// TIA Portal project "#13-J1200T(夹紧阀断电延时）" (V17)

(* hardware
DEVICE "S7-1200 station_1"  S7-1200 Station
   slot 0: "Rack_0"  S7-1200 Rack  Rack  V1.0
   slot 1: "PLC_1"  CPU 1215C DC/DC/DC  6ES7 215-1AG40-0XB0  V4.5
   slot 2: "DI 16x24VDC_1"  6ES7 221-1BH32-0XB0  V2.0
   slot 3: "DI 16x24VDC_2"  6ES7 221-1BH32-0XB0  V2.0
   slot 4: "DI 16x24VDC_3"  6ES7 221-1BH32-0XB0  V2.0
   slot 5: "DQ 16x24VDC_1"  SM 1222 DQ16 x 24VDC  6ES7 222-1BH32-0XB0  V2.0
   slot 101: "CM 1243-5"  CM 1243-5  6GK7 243-5DX30-0XE0  V1.3
DEVICE "ET 200SP station_1"  ET 200SP-Station
   slot 0: "机架_0"  Rack  6ES5 710-8MAx1
   slot 0: "IO device_1"  IM 155-6 PN ST  6ES7 155-6AU01-0BN0  V4.2
   slot 1: "DI 16x24VDC ST_1"  DI 16x24VDC ST  6ES7 131-6BH01-0BA0  V0.0
      slot 1: "DI 16x24VDC ST_1"  DI 16x24VDC ST
   slot 2: "DI 16x24VDC ST_6"  DI 16x24VDC ST  6ES7 131-6BH01-0BA0  V0.0
      slot 1: "DI 16x24VDC ST_6"  DI 16x24VDC ST
   slot 3: "DI 16x24VDC ST_5"  DI 16x24VDC ST  6ES7 131-6BH01-0BA0  V0.0
      slot 1: "DI 16x24VDC ST_5"  DI 16x24VDC ST
   slot 4: "DI 16x24VDC ST_4"  DI 16x24VDC ST  6ES7 131-6BH01-0BA0  V0.0
      slot 1: "DI 16x24VDC ST_4"  DI 16x24VDC ST
   slot 5: "DI 16x24VDC ST_3"  DI 16x24VDC ST  6ES7 131-6BH01-0BA0  V0.0
      slot 1: "DI 16x24VDC ST_3"  DI 16x24VDC ST
   slot 6: "DI 16x24VDC ST_2"  DI 16x24VDC ST  6ES7 131-6BH01-0BA0  V0.0
      slot 1: "DI 16x24VDC ST_2"  DI 16x24VDC ST
   slot 7: "DI 16x24VDC ST_7"  DI 16x24VDC ST  6ES7 131-6BH01-0BA0  V0.0
      slot 1: "DI 16x24VDC ST_7"  DI 16x24VDC ST
   slot 8: "DI 16x24VDC ST_8"  DI 16x24VDC ST  6ES7 131-6BH01-0BA0  V0.0
      slot 1: "DI 16x24VDC ST_8"  DI 16x24VDC ST
   slot 9: "DI 16x24VDC ST_9"  DI 16x24VDC ST  6ES7 131-6BH01-0BA0  V0.0
      slot 1: "DI 16x24VDC ST_9"  DI 16x24VDC ST
   slot 10: "DI 16x24VDC ST_10"  DI 16x24VDC ST  6ES7 131-6BH01-0BA0  V0.0
      slot 1: "DI 16x24VDC ST_10"  DI 16x24VDC ST
   slot 11: "DI 16x24VDC ST_11"  DI 16x24VDC ST  6ES7 131-6BH01-0BA0  V0.0
      slot 1: "DI 16x24VDC ST_11"  DI 16x24VDC ST
   slot 12: "DI 16x24VDC ST_12"  DI 16x24VDC ST  6ES7 131-6BH01-0BA0  V0.0
      slot 1: "DI 16x24VDC ST_12"  DI 16x24VDC ST
   slot 13: "DQ 16x24VDC/0.5A ST_2"  DQ 16x24VDC/0.5A ST  6ES7 132-6BH01-0BA0  V0.0
      slot 1: "DQ 16x24VDC/0.5A ST_2"  DQ 16x24VDC/0.5A ST
   slot 14: "DQ 16x24VDC/0.5A ST_1"  DQ 16x24VDC/0.5A ST  6ES7 132-6BH01-0BA0  V0.0
      slot 1: "DQ 16x24VDC/0.5A ST_1"  DQ 16x24VDC/0.5A ST
   slot 15: "服务器模块_1"  Server module  6ES7 193-6PA00-0AA0  V1.1
      slot 1: "服务器模块_1"  Server module
   slot 127: "BA 2xRJ45"  BA 2xRJ45  6ES7 193-6AR00-0AA0  V0.0
      slot 1: "Port_1"  X1 P1 R  6ES7 193-6AR00-0AA0  V0.0
      slot 2: "Port_2"  X1 P2 R  6ES7 193-6AR00-0AA0  V0.0
DEVICE "HMI_1"  TP900 Comfort
   slot 0: "HMI_1"  TP900 Comfort  6AV2 124-0JC01-0AX0  15.1.0.0
   slot 1: "HMI_RT_1"  TP900 Comfort  6AV2 124-0JC01-0AX0  15.1.0.0
   slot 5: "HMI_1.IE_CP_1"  PROFINET Interface  15.0.1.0
      slot 1: "PROFINET Interface_1"  PROFINET Interface
         slot 1: "Port_1"  Port
         slot 2: "Port_2"  Port
   slot 7: "HMI_1.MPI/DP_CP_1"  MPI/DP Interface  15.0.1.0
DEVICE "GSD device_2"  GSD.Device
   slot 0: "机架_0"  Rail
   slot 0: "HENGLIANGBIANMAQI"  P+F  Encoder  4.0
DEVICE "GSD device_1"  GSD.Device
   slot 0: "机架_0"  Rail
   slot 0: "滑块站"  P+F  Encoder  4.0
*)

// ===== PLC "PLC_1"  CPU 1215C DC/DC/DC =====

VAR_GLOBAL   // PLC tag table "默认变量表"
   "Tag_1" AT %I0.0 : Bool;
   "Tag_2" AT %I0.1 : Bool;
   "Tag_3" AT %I0.2 : Bool;
   "Tag_4" AT %I0.3 : Bool;
   "Tag_5" AT %I0.4 : Bool;
   "Tag_6" AT %I0.5 : Bool;
   "Tag_7" AT %I0.6 : Bool;
   "Tag_8" AT %I0.7 : Bool;
   "Tag_9" AT %I1.0 : Bool;
   "Tag_10" AT %I1.1 : Bool;
   "Tag_11" AT %I1.2 : Bool;
   "Tag_12" AT %I1.3 : Bool;
   "Tag_13" AT %I1.4 : Bool;
   "Tag_14" AT %I1.5 : Bool;
   "润滑空开" AT %I2.0 : Bool;
   "润滑电机1过载" AT %I2.1 : Bool;
   "Tag_17" AT %I2.4 : Bool;
   "急停KA12" AT %I2.5 : Bool;
   "双阀反馈1" AT %I2.6 : Bool;
   "双阀故障" AT %I3.2 : Bool;
   "滑块空开" AT %I3.3 : Bool;
   "滑块调整防粘连" AT %I3.4 : Bool;
   "Tag_23" AT %I3.5 : Bool;
   "气垫调整空开" AT %I3.6 : Bool;
   "润滑电机2过载_" AT %I2.2 : Bool;
   "润滑电机3过载_" AT %I2.3 : Bool;
   "双阀反馈2" AT %I2.7 : Bool;
   "双阀反馈3" AT %I3.0 : Bool;
   "双阀反馈4" AT %I3.1 : Bool;
   "气垫调整防粘连" AT %I3.7 : Bool;
   "右栅栏空开" AT %I4.0 : Bool;
   "栅栏空开防粘连" AT %I4.1 : Bool;
   "安全栓" AT %I4.2 : Bool;
   "油箱加热触点" AT %I4.3 : Bool;
   "电柜冷却触点" AT %I4.4 : Bool;
   "电机风机启动" AT %I4.5 : Bool;
   "Tag_21" AT %I4.6 : Bool;
   "Tag_22" AT %I4.7 : Bool;
   "Tag_23(1)" AT %I5.0 : Bool;
   "Tag_24" AT %I5.1 : Bool;
   "Tag_25" AT %I5.2 : Bool;
   "Tag_26" AT %I5.3 : Bool;
   "Tag_27" AT %I5.4 : Bool;
   "Tag_28" AT %I5.5 : Bool;
   "Tag_29" AT %I5.6 : Bool;
   "Tag_30" AT %I5.7 : Bool;
   "Tag_31" AT %I6.0 : Bool;
   "Tag_32" AT %I6.1 : Bool;
   "Tag_33" AT %I6.2 : Bool;
   "Tag_34" AT %I6.3 : Bool;
   "Tag_35" AT %I6.4 : Bool;
   "Tag_36" AT %I6.5 : Bool;
   "Tag_37" AT %I6.6 : Bool;
   "Tag_38" AT %I6.7 : Bool;
   "Tag_39" AT %I7.0 : Bool;
   "Tag_40" AT %I7.1 : Bool;
   "Tag_41" AT %I7.2 : Bool;
   "Tag_42" AT %I7.3 : Bool;
   "Tag_43" AT %I7.4 : Bool;
   "Tag_44" AT %I7.5 : Bool;
   "Tag_45" AT %I7.6 : Bool;
   "Tag_46" AT %I7.7 : Bool;
   "气垫手动润滑" AT %I10.0 : Bool;
   "平衡缸手动润滑" AT %I10.1 : Bool;
   "润滑电机启动" AT %I10.2 : Bool;
   "润滑电机停止" AT %I10.3 : Bool;
   "主电机停止" AT %I10.4 : Bool;
   "主电机启动" AT %I10.5 : Bool;
   "微调正反" AT %I10.6 : Bool;
   "微调开动" AT %I10.7 : Bool;
   "气垫调整" AT %I11.0 : Bool;
   "滑块调整" AT %I11.1 : Bool;
   "行程" AT %I11.2 : Bool;
   "模具更换" AT %I11.3 : Bool;
   "微调(1)" AT %I11.4 : Bool;
   "连续" AT %I11.5 : Bool;
   "单次" AT %I11.6 : Bool;
   "寸动" AT %I11.7 : Bool;
   "数据编辑" AT %I12.0 : Bool;
   "寸动1" AT %I12.1 : Bool;
   "寸动2" AT %I12.2 : Bool;
   "连续预置" AT %I12.3 : Bool;
   "停上死点" AT %I12.4 : Bool;
   "故障复位" AT %I12.5 : Bool;
   "液压保护实验" AT %I12.6 : Bool;
   "液压保护重调" AT %I12.7 : Bool;
   "滑块向上" AT %I13.0 : Bool;
   "滑块向下" AT %I13.1 : Bool;
   "滑块调整手动/自动" AT %I13.2 : Bool;
   "模具夹紧/松开" AT %I13.3 : Bool;
   "工作台夹紧/放松" AT %I13.4 : Bool;
   "备用(1)" AT %I13.5 : Bool;
   "油箱加热启动" AT %I13.6 : Bool;
   "油箱加热停止" AT %I13.7 : Bool;
   "平衡缸压力手动/自动" AT %I14.0 : Bool;
   "气垫压力手动/自动" AT %I14.1 : Bool;
   "气垫快排" AT %I14.2 : Bool;
   "气垫调整手动/自动" AT %I14.3 : Bool;
   "气垫向上" AT %I14.4 : Bool;
   "气垫向下" AT %I14.5 : Bool;
   "安全栅栏向上" AT %I14.6 : Bool;
   "安全栅栏向下" AT %I14.7 : Bool;
   "低油位" AT %I15.0 : Bool;
   "高油位" AT %I15.1 : Bool;
   "低油压1" AT %I15.2 : Bool;
   "低油压2" AT %I15.3 : Bool;
   "低油压3" AT %I15.4 : Bool;
   "高油压1" AT %I15.5 : Bool;
   "高油压2" AT %I15.6 : Bool;
   "高油压3" AT %I15.7 : Bool;
   "左前移动闭点1" AT %I16.0 : Bool;
   "左前移动闭点2" AT %I16.1 : Bool;
   "左前移动开点" AT %I16.2 : Bool;
   "左前移动检测" AT %I16.3 : Bool;
   "左后移动闭点1" AT %I16.4 : Bool;
   "左后移动闭点2" AT %I16.5 : Bool;
   "左后移动开点" AT %I16.6 : Bool;
   "左后移动检测" AT %I16.7 : Bool;
   "右前移动短接1" AT %I17.0 : Bool;
   "右前移动短接2" AT %I17.1 : Bool;
   "右前移动短接3" AT %I17.2 : Bool;
   "右前移动短接4" AT %I17.3 : Bool;
   "右后移动短接1" AT %I17.4 : Bool;
   "右后移动短接2" AT %I17.5 : Bool;
   "右后移动短接3" AT %I17.6 : Bool;
   "右后移动短接4" AT %I17.7 : Bool;
   "备用" AT %I18.0 : Bool;
   "梯子开关" AT %I18.1 : Bool;
   "飞轮制动1" AT %I18.2 : Bool;
   "飞轮制动2" AT %I18.3 : Bool;
   "温度保护" AT %I18.4 : Bool;
   "主接触器" AT %I18.5 : Bool;
   "磁场电源" AT %I18.6 : Bool;
   "同步电源" AT %I18.7 : Bool;
   "装置风扇" AT %I19.0 : Bool;
   "风机" AT %I19.1 : Bool;
   "装置正常" AT %I19.2 : Bool;
   "电流保护" AT %I19.3 : Bool;
   "气垫润滑高压" AT %I19.4 : Bool;
   "过滤器堵塞1" AT %I19.5 : Bool;
   "过滤器堵塞2" AT %I19.6 : Bool;
   "过滤器堵塞3" AT %I19.7 : Bool;
   "润滑检测1" AT %I20.0 : Bool;
   "润滑检测2" AT %I20.1 : Bool;
   "润滑检测3" AT %I20.2 : Bool;
   "润滑检测4" AT %I20.3 : Bool;
   "润滑检测5" AT %I20.4 : Bool;
   "润滑检测6" AT %I20.5 : Bool;
   "润滑检测7" AT %I20.6 : Bool;
   "润滑检测8" AT %I20.7 : Bool;
   "润滑检测9" AT %I21.0 : Bool;
   "备用(2)" AT %I21.1 : Bool;
   "离合器压力" AT %I21.2 : Bool;
   "制动器压力" AT %I21.3 : Bool;
   "凸轮1" AT %I21.4 : Bool;
   "凸轮2" AT %I21.5 : Bool;
   "凸轮3" AT %I21.6 : Bool;
   "凸轮4" AT %I21.7 : Bool;
   "灯测试" AT %I22.0 : Bool;
   "蜂鸣器按钮" AT %I22.1 : Bool;
   "自动化气源测试" AT %I22.2 : Bool;
   "Tag_146" AT %I22.3 : Bool;
   "液压保护压力" AT %I22.4 : Bool;
   "卸荷限位" AT %I22.5 : Bool;
   "Tag_149" AT %I22.6 : Bool;
   "滑块上限" AT %I22.7 : Bool;
   "滑块下限" AT %I23.0 : Bool;
   "滑块调整过扭矩" AT %I23.1 : Bool;
   "Tag_153" AT %I23.2 : Bool;
   "Tag_154" AT %I23.3 : Bool;
   "气垫上限" AT %I23.4 : Bool;
   "气垫下限" AT %I23.5 : Bool;
   "Tag_157" AT %I23.6 : Bool;
   "Tag_158" AT %I23.7 : Bool;
   "Tag_159" AT %I24.0 : Bool;
   "Tag_160" AT %I24.1 : Bool;
   "安全栅栏上限位" AT %I24.2 : Bool;
   "安全栅栏下限位" AT %I24.3 : Bool;
   "气垫落到位" AT %I24.4 : Bool;
   "温度开关" AT %I24.5 : Bool;
   "工作台夹紧" AT %I24.6 : Bool;
   "工作台放松" AT %I24.7 : Bool;
   "Tag_167" AT %I25.0 : Bool;
   "平衡缸压力" AT %I25.1 : Bool;
   "工作台夹紧压力" AT %I25.2 : Bool;
   "工作台放松压力" AT %I25.3 : Bool;
   "Tag_171" AT %I25.4 : Bool;
   "Tag_172" AT %I25.5 : Bool;
   "Tag_173" AT %I25.6 : Bool;
   "Tag_174" AT %I25.7 : Bool;
   "Tag_175" AT %I26.0 : Bool;
   "Tag_176" AT %I26.1 : Bool;
   "工作台前落到位" AT %I26.2 : Bool;
   "工作台后落到位" AT %I26.3 : Bool;
   "光电保护开" AT %I26.4 : Bool;
   "光电保护1" AT %I26.5 : Bool;
   "光电保护2" AT %I26.6 : Bool;
   "光电保护3" AT %I26.7 : Bool;
   "光电保护4" AT %I27.0 : Bool;
   "高度保护复位" AT %I27.1 : Bool;
   "防重复3231" AT %I27.2 : Bool;
   "防重复检测3232" AT %I27.3 : Bool;
   "吨位监控" AT %I27.5 : Bool;
   "光电保护角度3235" AT %I27.6 : Bool;
   "Tag_190" AT %I27.7 : Bool;
   "Tag_191" AT %I28.0 : Bool;
   "Tag_192" AT %I28.1 : Bool;
   "Tag_193" AT %I28.2 : Bool;
   "Tag_194" AT %I28.3 : Bool;
   "Tag_195" AT %I28.4 : Bool;
   "Tag_196" AT %I28.5 : Bool;
   "Tag_197" AT %I28.6 : Bool;
   "Tag_198" AT %I28.7 : Bool;
   "Tag_199" AT %I29.0 : Bool;
   "Tag_200" AT %I29.1 : Bool;
   "Tag_201" AT %I29.2 : Bool;
   "Tag_202" AT %I29.3 : Bool;
   "Tag_203" AT %I29.4 : Bool;
   "Tag_204" AT %I29.5 : Bool;
   "Tag_205" AT %I29.6 : Bool;
   "Tag_206" AT %I29.7 : Bool;
   "Tag_207" AT %I30.0 : Bool;
   "Tag_208" AT %I30.1 : Bool;
   "Tag_209" AT %I30.2 : Bool;
   "Tag_210" AT %I30.3 : Bool;
   "Tag_211" AT %I30.4 : Bool;
   "Tag_212" AT %I30.5 : Bool;
   "Tag_213" AT %I30.6 : Bool;
   "Tag_214" AT %I30.7 : Bool;
   "Tag_215" AT %I31.0 : Bool;
   "Tag_216" AT %I31.1 : Bool;
   "Tag_217" AT %I31.2 : Bool;
   "Tag_218" AT %I31.3 : Bool;
   "Tag_219" AT %I31.4 : Bool;
   "Tag_220" AT %I31.5 : Bool;
   "Tag_221" AT %I31.6 : Bool;
   "Tag_222" AT %I31.7 : Bool;
   "Tag_223" AT %I32.0 : Bool;
   "Tag_224" AT %I32.1 : Bool;
   "Tag_225" AT %I32.2 : Bool;
   "Tag_226" AT %I32.3 : Bool;
   "Tag_227" AT %I32.4 : Bool;
   "Tag_228" AT %I32.5 : Bool;
   "Tag_229" AT %I32.6 : Bool;
   "Tag_230" AT %I32.7 : Bool;
   "Tag_231" AT %I33.0 : Bool;
   "Tag_232" AT %I33.1 : Bool;
   "Tag_233" AT %I33.2 : Bool;
   "Tag_234" AT %I33.3 : Bool;
   "Tag_235" AT %I33.4 : Bool;
   "Tag_236" AT %I33.5 : Bool;
   "Tag_237" AT %I33.6 : Bool;
   "Tag_238" AT %I33.7 : Bool;
   "横梁编码器" AT %ID68 : DWord;
   "滑块编码器" AT %ID72 : DInt;
   "Tag_15" AT %Q0.0 : Bool;
   "Tag_16" AT %Q0.1 : Bool;
   "Tag_17(1)" AT %Q0.2 : Bool;
   "Tag_18" AT %Q0.3 : Bool;
   "Tag_19" AT %Q0.4 : Bool;
   "Tag_20" AT %Q0.5 : Bool;
   "Tag_21(1)" AT %Q0.6 : Bool;
   "Tag_22(1)" AT %Q0.7 : Bool;
   "Tag_23(2)" AT %Q1.0 : Bool;
   "Tag_24(1)" AT %Q1.1 : Bool;
   "KA8主电机主接触器" AT %Q2.0 : Bool;
   "KA9主电机正转启动" AT %Q2.1 : Bool;
   "KA10" AT %Q2.2 : Bool;
   "KA11" AT %Q2.3 : Bool;
   "KA12" AT %Q2.4 : Bool;
   "润滑启动(1)" AT %Q2.5 : Bool;
   "气垫调整防粘连(1)" AT %Q2.6 : Bool;
   "气垫向上(2)" AT %Q2.7 : Bool;
   "气垫向下(2)" AT %Q3.0 : Bool;
   "右栅栏防粘连(1)" AT %Q3.1 : Bool;
   "右栅栏向上(1)" AT %Q3.2 : Bool;
   "右栅栏向下(1)" AT %Q3.3 : Bool;
   "润滑油加热(1)" AT %Q3.4 : Bool;
   "滑块调整防粘连(2)" AT %Q3.5 : Bool;
   "滑块向上调整(1)" AT %Q3.6 : Bool;
   "滑块向下调整(1)" AT %Q3.7 : Bool;
   "上死点指示(1)" AT %Q10.0 : Bool;
   "模具放松指示" AT %Q10.1 : Bool;
   "润滑正常指示" AT %Q10.2 : Bool;
   "滤油器堵塞指示" AT %Q10.3 : Bool;
   "油箱油位高指示" AT %Q10.4 : Bool;
   "主电机运行指示" AT %Q10.5 : Bool;
   "液压保护正常指示" AT %Q10.6 : Bool;
   "气垫 落到位指示" AT %Q10.7 : Bool;
   "连续预置指示" AT %Q11.0 : Bool;
   "警铃" AT %Q11.1 : Bool;
   "设备故障指示" AT %Q11.2 : Bool;
   "光电保护指示" AT %Q11.3 : Bool;
   "下死点指示" AT %Q11.4 : Bool;
   "工作台就位夹紧指示" AT %Q11.5 : Bool;
   "工作台放松指示" AT %Q11.6 : Bool;
   "油箱加热指示" AT %Q11.7 : Bool;
   "制动器阀" AT %Q12.0 : Bool;
   "离合器阀1" AT %Q12.1 : Bool;
   "离合器阀2" AT %Q12.2 : Bool;
   "飞轮制动阀" AT %Q12.3 : Bool;
   "平衡缸润滑阀" AT %Q12.4 : Bool;
   "液压保护气源阀" AT %Q12.5 : Bool;
   "液压保护气动泵阀" AT %Q12.6 : Bool;
   "气垫快排阀" AT %Q12.7 : Bool;
   "工作台夹紧阀" AT %Q13.0 : Bool;
   "工作台放松阀" AT %Q13.1 : Bool;
   "气垫润滑阀" AT %Q13.2 : Bool;
   "Tag_95" AT %Q13.3 : Bool;
   "Tag_96" AT %Q13.4 : Bool;
   "Tag_97" AT %Q13.5 : Bool;
   "Tag_98" AT %Q13.6 : Bool;
   "Tag_99" AT %Q13.7 : Bool;
   "Tag_100" AT %Q14.0 : Bool;
   "Tag_101" AT %Q14.1 : Bool;
   "Tag_102" AT %Q14.2 : Bool;
   "Tag_103" AT %Q14.3 : Bool;
   "Tag_104" AT %Q14.4 : Bool;
   "Tag_105" AT %Q14.5 : Bool;
   "Tag_106" AT %Q14.6 : Bool;
   "Tag_107" AT %Q14.7 : Bool;
   "润滑电机过载" AT %M300.0 : Bool;
   "润滑油压低" AT %M300.1 : Bool;
   "润滑高油压" AT %M300.2 : Bool;
   "润滑故障分钟检测" AT %M400.0 : Bool;
   "润滑低油位" AT %M300.3 : Bool;
   "润滑高油位" AT %M300.4 : Bool;
   "润滑故障" AT %M500.0 : Bool;
   "主电机关断延时" AT %M320.1 : Bool;
   "滑块调整条件" AT %M330.0 : Bool;
   "寸动条件1" AT %M7008.0 : Bool;
   "寸动条件2" AT %M7008.1 : Bool;
   "液压保护正常" AT %M7010.0 : Bool;
   "10度" AT %M200.0 : Bool;
   "20度" AT %M200.1 : Bool;
   "30度" AT %M200.2 : Bool;
   "40度" AT %M200.3 : Bool;
   "50" AT %M200.4 : Bool;
   "60" AT %M200.5 : Bool;
   "70" AT %M200.6 : Bool;
   "80" AT %M200.7 : Bool;
   "90" AT %M201.0 : Bool;
   "100" AT %M201.1 : Bool;
   "110" AT %M201.2 : Bool;
   "120" AT %M201.3 : Bool;
   "130" AT %M201.4 : Bool;
   "140" AT %M201.5 : Bool;
   "150" AT %M201.6 : Bool;
   "160" AT %M201.7 : Bool;
   "170" AT %M202.0 : Bool;
   "180" AT %M202.1 : Bool;
   "190" AT %M202.2 : Bool;
   "200" AT %M202.3 : Bool;
   "210" AT %M202.4 : Bool;
   "220" AT %M202.5 : Bool;
   "230" AT %M202.6 : Bool;
   "240" AT %M202.7 : Bool;
   "250" AT %M203.0 : Bool;
   "260" AT %M203.1 : Bool;
   "270" AT %M203.2 : Bool;
   "280" AT %M203.3 : Bool;
   "290" AT %M203.4 : Bool;
   "300" AT %M203.5 : Bool;
   "310" AT %M203.6 : Bool;
   "320" AT %M203.7 : Bool;
   "330" AT %M204.0 : Bool;
   "340" AT %M204.1 : Bool;
   "350" AT %M204.2 : Bool;
   "360" AT %M204.3 : Bool;
   "上死点" AT %M204.4 : Bool;
   "制动监控" AT %M204.5 : Bool;
   "下死点" AT %M204.6 : Bool;
   "单次返回" AT %M204.7 : Bool;
   "光电保护位置" AT %M205.0 : Bool;
   "编码器闭点监控" AT %M14.7 : Bool;
   "单次开始" AT %M14.4 : Bool;
   "编码器开点监控" AT %M15.0 : Bool;
   "编码器故障" AT %M15.1 : Bool;
   "上死点指示" AT %M0.0 : Bool;
   "下死点指示(1)" AT %M0.1 : Bool;
   "滑块软限位上" AT %M15.5 : Bool;
   "上调整设定值" AT %M15.7 : Bool;
   "滑块软限位下" AT %M15.6 : Bool;
   "滑块调整自动向下" AT %M16.1 : Bool;
   "微调反转" AT %M0.2 : Bool;
   "滑块调整自动向上" AT %M16.0 : Bool;
   "滑块调整自动选择" AT %M16.2 : Bool;
   "微调正转" AT %M0.3 : Bool;
   "行程允许" AT %M14.0 : Bool;
   "寸动允许" AT %M14.1 : Bool;
   "寸动开始" AT %M14.2 : Bool;
   "单次允许" AT %M14.3 : Bool;
   "双手开点监测" AT %M11.0 : Bool;
   "双手闭点监测" AT %M11.1 : Bool;
   "急停故障" AT %M6.0 : Bool;
   "润滑次数检测" AT %M11.2 : Bool;
   "润滑频次故障" AT %M11.3 : Bool;
   "单次返回3233" AT %I27.4 : Bool;
   "重复故障" AT %M19.1 : Bool;
   "计数开始" AT %M20.0 : Bool;
   "计数清零" AT %M20.1 : Bool;
   "间歇润滑时间" AT %M19.3 : Bool;
   "Tag_47" AT %MB10 : Byte;
   "Tag_48" AT %MD10 : DWord;
END_VAR

VAR_GLOBAL CONSTANT   // PLC tag table "默认变量表"
   "无(1)" : Pip := 65535;
   "自动更新(1)" : Pip := 0;
   "PIP 1(1)" : Pip := 1;
   "PIP 2(1)" : Pip := 2;
   "PIP 3(1)" : Pip := 3;
   "PIP 4(1)" : Pip := 4;
   "PIP OB 伺服(1)" : Pip := 32768;
   "Local~MC(1)" : Hw_SubModule := 51;
   "Local~Common(1)" : Hw_SubModule := 50;
   "Local~Device(1)" : Hw_Device := 32;
   "Local~Configuration(1)" : Hw_SubModule := 33;
   "Local~Exec(1)" : Hw_SubModule := 52;
   "Local(1)" : Hw_SubModule := 49;
   "Local~PROFINET_接口_1(1)" : Hw_Interface := 64;
   "Local~PROFINET_接口_1~端口_1(1)" : Hw_Interface := 65;
   "Local~HSC_1(1)" : Hw_Hsc := 257;
   "Local~HSC_2(1)" : Hw_Hsc := 258;
   "Local~HSC_3(1)" : Hw_Hsc := 259;
   "Local~HSC_4(1)" : Hw_Hsc := 260;
   "Local~HSC_5(1)" : Hw_Hsc := 261;
   "Local~HSC_6(1)" : Hw_Hsc := 262;
   "Local~AI_2_1" : Hw_SubModule := 263;
   "Local~DI_14_DQ_10_1(1)" : Hw_SubModule := 264;
   "Local~Pulse_1(1)" : Hw_Pwm := 265;
   "Local~Pulse_2(1)" : Hw_Pwm := 266;
   "Local~Pulse_3(1)" : Hw_Pwm := 267;
   "Local~Pulse_4(1)" : Hw_Pwm := 268;
   "Local~CM_1243-5~DP_接口(1)" : Hw_Interface := 269;
   "Local~CM_1243-5(1)" : Hw_SubModule := 271;
   "Local~PROFINET_IO-System(1)" : Hw_IoSystem := 272;
   "Local~DP-Mastersystem(1)" : Hw_IoSystem := 273;
   "Local~DI_16x24VDC_1(1)" : Hw_SubModule := 291;
   "Local~DI_16x24VDC_2(1)" : Hw_SubModule := 292;
   "Local~DQ_16x24VDC_1(1)" : Hw_SubModule := 293;
   "立柱右前操作站~Head" : Hw_Interface := 288;
   "立柱右前操作站~DPSlave" : Hw_DpSlave := 286;
   "立柱右前操作站~DI_32x24VDC_1" : Hw_SubModule := 289;
   "立柱右前操作站~AI_8x12BIT_1" : Hw_SubModule := 294;
   "立柱右前操作站~DI_32x24VDC_2" : Hw_SubModule := 295;
   "立柱右前操作站~DI_32x24VDC_3" : Hw_SubModule := 296;
   "立柱右前操作站~DI_32x24VDC_4" : Hw_SubModule := 297;
   "立柱右前操作站~DO_32x24VDC_0_5A_2" : Hw_SubModule := 299;
   "立柱右前操作站~DO_16x24VDC_0_5A_1" : Hw_SubModule := 290;
   "立柱右前操作站~DI_16x24VDC_1" : Hw_SubModule := 274;
   "横梁站~Head(1)" : Hw_Interface := 280;
   "横梁站~DPSlave(1)" : Hw_DpSlave := 278;
   "横梁站~P+F_Version_2_1_Singleturn_1(1)" : Hw_SubModule := 281;
   "OB_Main(1)" : OB_PCYCLE := 1;
   "OB_Cyclic interrupt" : OB_Cyclic := 30;
   "OB_RackStationFailure" : OB_Any := 86;
   "OB_Startup" : OB_STARTUP := 100;
   "滑块站~Head(1)" : Hw_Interface := 277;
   "滑块站~DPSlave(1)" : Hw_DpSlave := 275;
   "滑块站~32_Bit_Class_2_+_Speed_2_1" : Hw_SubModule := 282;
   "滑块站~32_Bit_Class_2_+_Speed_2_2" : Hw_SubModule := 283;
END_VAR

VAR_GLOBAL   // PLC tag table "变量表_1"
   "主电机启动条件" AT %M800.1 : Bool;
   "产量完成" AT %M800.0 : Bool;
END_VAR

TYPE "用户数据类型_1"
VERSION : 0.1
   STRUCT
      Element_1 : Bool;
   END_STRUCT;
END_TYPE

// folder: 4.1_Line_Operation

TYPE "Operation_Mode"
VERSION : 0.1
   STRUCT
      Auto : Bool;
      Auto_Sim : Bool;
      APC : Bool;
      ATC : Bool;
      Man : Bool;
      Setup : Bool;
      工作模式 : UInt;
      零件表 : UInt;
   END_STRUCT;
END_TYPE

TYPE "4.1_Line_Operation"
VERSION : 0.1
   STRUCT
      Mode_Act : "Operation_Mode";
      Mode_Seting : "Operation_Mode";
      Recipes_Operation : "HMI_Recipe";
      HMI : Array[1..10] of "HMI_State";
   END_STRUCT;
END_TYPE

TYPE "HMI_Recipe"
VERSION : 0.1
   STRUCT
      Recipe : Struct
         Clear : Bool;
         Load : Bool;
         Save : Bool;
         Edit_No : Int;
         Recipe_Edit_Auth : Bool;
         Recipe_Edit_Wizard : Int;
         Load_Active : Bool;
         Save_Active : Bool;
         ii : Int;
         Load_Timer : IEC_TIMER;
         Save_Timer : IEC_TIMER;
      END_STRUCT;
      RecipeExport : Struct
         Done : Bool;
         Busy : Bool;
         Error : Bool;
         Status : Word;
      END_STRUCT;
      RecipeImport : Struct
         Done : Bool;
         Busy : Bool;
         Error : Bool;
         Status : Word;
      END_STRUCT;
   END_STRUCT;
END_TYPE

TYPE "HMI_State"
VERSION : 0.1
   STRUCT
      Command : Struct
         Doub_Part_Dropped_Mem : Bool;
         Part_Dropped_Mem : Bool;
         Part_Picker_Mem : Bool;
         Part_Done_Mem : Bool;
         Optim_Auth : Bool;
         Part_No_Chg_Auth : Bool;
      END_STRUCT;
      State : Struct
         Doub_Part_Dropped_Mem_1 : Bool;
         Part_Dropped_Mem_1 : Bool;
         Part_Picker_Mem_1 : Bool;
         Part_Done_Mem_1 : Bool;
      END_STRUCT;
   END_STRUCT;
END_TYPE

// folder: (top level)

DATA_BLOCK "横梁编码器 _DB"   // DB15
{ S7_Optimized_Access := 'TRUE' }
VERSION : 0.1
   VAR
      "0.0" : Struct
         "+0.0" : DWord;
         "+4.0" : DWord;
         "+8.0" : DWord;
         "+12.0" : DWord;
      END_STRUCT;
      横梁 : Int;
      滑块 : Int;
      滑块_1 : DWord;
      "+0.3" : Int;
      "+0.4" : Int;
      "+0.5" : Int;
      "+0.6" : Int;
      "+0.7" : Int;
   END_VAR
   VAR RETAIN
      "+0.8" : Int;
   END_VAR
   VAR
      "+0.9" : Int;
      "+0.10" : Int;
      "0.11" : Real;
      平衡器分油器检测 : Int;
      横梁分油器检测 : Int;
      滑块分油器检测 : Int;
      气垫分油器检测 : Int;
      "+0.15" : Int;
      "+0.16" : Int;
      "+0.17" : Int;
      "+0.18" : Int;
      "+0.19" : Int;
      "+0.20" : Int;
      "+0.21" : Int;
      "+0.22" : Int;
      "+0.23" : Int;
      "+0.24" : Int;
      "+0.25" : Int;
      "+0.26" : Int;
      "+0.27" : Int;
      "+0.28" : Int;
      "+0.29" : Int;
      "+0.30" : Int;
      平衡器打油次数 : Int;
      主分油器打油次数 : Int;
      滑块打油次数 : Int;
      气点垫打油次数 : Int;
      "+0.35" : Int;
      "+0.36" : Int;
      "+0.37" : Int;
      "+0.38" : Int;
      "+0.39" : Int;
      "+0.40" : Int;
      "+0.41" : Int;
      "+0.42" : Int;
      "+0.43" : Int;
      "+0.44" : Int;
      "+0.45" : Int;
      "+0.46" : Int;
      "+0.47" : Int;
      "+0.48" : Int;
   END_VAR
   VAR RETAIN
      AI : Array[0..10] of DInt;
      D : Array[0..10] of Real;
   END_VAR
   VAR
      AQD : Real;
      产量设定 : Int;
      D107 : Real;
   END_VAR
BEGIN
END_DATA_BLOCK

DATA_BLOCK "滑块编码器_DB"   // DB16
{ S7_Optimized_Access := 'TRUE' }
VERSION : 0.1
   VAR
      "0.0" : Struct
         "+0.0" : DWord;
         "+4.0" : DWord;
         "+8.0" : DWord;
         "+12.0" : DWord;
      END_STRUCT;
      横梁编码器 : Int;
      滑块编码器 : DInt;
      气垫编码器1 : DWord;
      气垫编码器2 : DWord;
      平衡器压力显示_3 : Int;
      电子凸轮编码器 : Int;
      "+0.5" : Real;
      电子凸轮编码器显示 : Int;
      "+0.7" : DInt;
      "+0.8" : Int;
      "+0.9" : Real;
      "+0.10_1" : Int;
      "+0.11" : Int;
      "+0.12" : Int;
      "+0.13" : Int;
      "+0.10" : Int;
      平衡器分油器检测 : Int;
      横梁分油器检测 : Int;
      滑块分油器检测 : Int;
      气垫分油器检测 : Int;
      "+0.15" : Int;
      "+0.16" : Int;
      "+0.17" : Int;
      "+0.18" : Int;
      "+0.19" : Int;
      "+0.20" : Int;
      "+0.21" : Int;
      "+0.22" : Int;
      "+0.23" : Int;
      "+0.24" : Int;
      "+0.25" : Int;
      "+0.26" : Int;
      "+0.27" : Int;
      "+0.28" : Int;
      "+0.29" : Int;
      "+0.30" : Int;
      平衡器打油次数 : Int;
      主分油器打油次数 : Int;
      滑块打油次数 : Int;
      气点垫打油次数 : Int;
      "+0.35" : Int;
      "+0.36" : Int;
      平衡器压力显示_2 : Real;
      平衡器压力显示_1 : Real;
      "+0.39" : Int;
      "+0.40" : Real;
      "+0.41" : Real;
      气垫模拟量 : Int;
      气垫模拟量_1 : Real;
      气垫模拟量_2 : Real;
      "+0.45" : DInt;
      "+0.46" : Int;
      "+0.47" : Real;
      "+0.48" : Int;
   END_VAR
   VAR RETAIN
      AI : Array[0..10] of DInt;
      D : Array[0..20] of Real;
   END_VAR
   VAR
      平衡器压力显示 : Real;
      AQD2 : Real;
      气垫模拟量显示1 : Real;
      气垫模拟量显示2 : Real;
      平衡器设置压力 : Real;
      气垫1压力设置 : Real;
      气垫2压力设置 : Real;
      D100 : Real;
      D101 : Int;
      D102 : Int;
      D103 : Real;
      D104 : Real;
      D105 : Real;
      D106 : Real;
      D107 : Int;
      D108 : Real;
      D109 : Real;
   END_VAR
   VAR RETAIN
      设置产量 : Int;
      当前产量 : Int;
      滑块位置 : Int;
   END_VAR
   VAR
      气垫位置 : Int;
   END_VAR
   VAR RETAIN
      D200 : DInt;
      D201 : Int;
   END_VAR
BEGIN
END_DATA_BLOCK

DATA_BLOCK "计时器"   // DB20
{ S7_Optimized_Access := 'TRUE' }
VERSION : 0.1
   VAR
      润滑检测延时 : IEC_TIMER;
      编码器闭店监控延时 : IEC_TIMER;
      编码器开点监控延时 : IEC_TIMER;
      主电机指示延时 : IEC_TIMER;
      润滑次数检测延时 : IEC_TIMER;
      平衡缸自动润滑计时 : IEC_TIMER;
      气垫自动润滑计时 : IEC_TIMER;
      平衡缸自动润滑间隔 : IEC_TIMER;
      气垫自动润滑间隔 : IEC_TIMER;
      夹紧阀断电延时 : IEC_TIMER;
   END_VAR
BEGIN
END_DATA_BLOCK

DATA_BLOCK "计数器"   // DB21
{ S7_Optimized_Access := 'TRUE' }
VERSION : 0.1
   VAR
      润滑次数检测 : IEC_COUNTER;
   END_VAR
   VAR RETAIN
      产品计数 : IEC_COUNTER;
   END_VAR
BEGIN
END_DATA_BLOCK

DATA_BLOCK "断电保持数据"   // DB30
{ S7_Optimized_Access := 'TRUE' }
VERSION : 0.1
   VAR RETAIN
      当前产量 : Int := 0;
      目标产量 : Int;
   END_VAR
BEGIN
END_DATA_BLOCK

// folder: 04_HMI_Comand_Config

DATA_BLOCK "Line_OP"   // DB10
{ S7_Optimized_Access := 'TRUE' }
VERSION : 0.1
BEGIN
END_DATA_BLOCK

// folder: (top level)

FUNCTION "10-润滑启动" : Void   // FC10, LAD
{ S7_Optimized_Access := 'TRUE' }
VERSION : 0.1
   VAR_TEMP   // added for the SCL form of the ladder/FBD networks
      _w1 : Bool;
   END_VAR
BEGIN

REGION Network 1
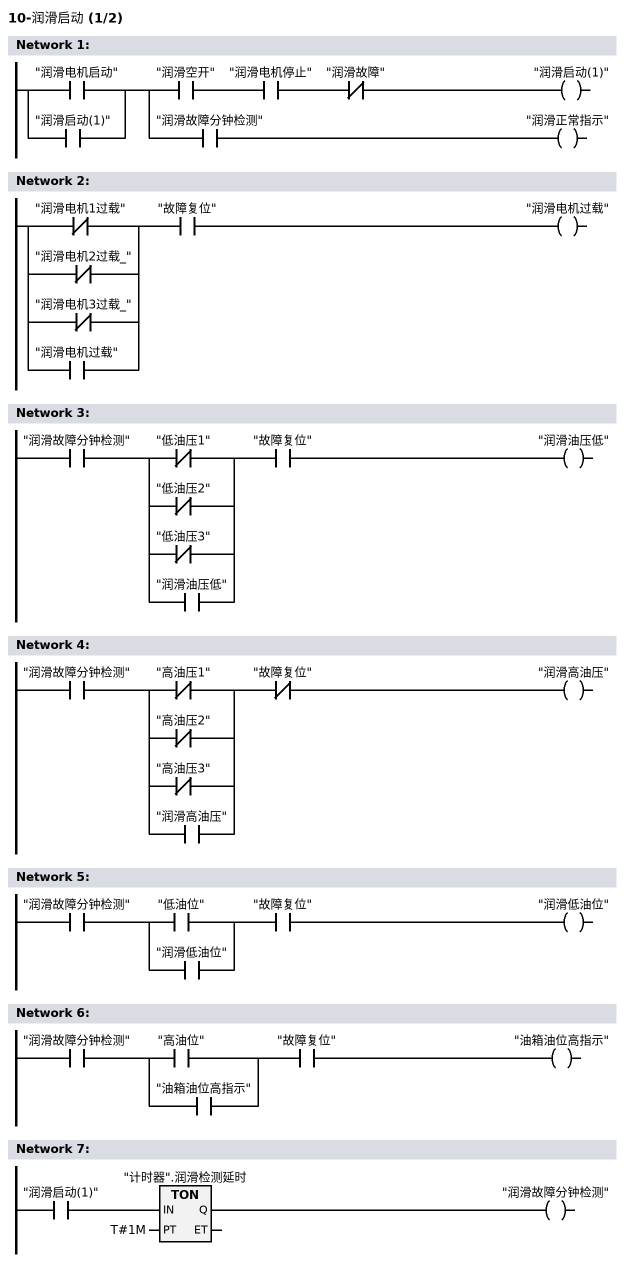
   RUNG wire#powerrail
      Contact( "润滑电机启动" )
      wire#w1
      Contact( "润滑空开" )
      Contact( "润滑电机停止" )
      I_Contact( "润滑故障" )
      Coil( "润滑启动(1)" )
   END_RUNG
   RUNG wire#powerrail
      Contact( "润滑启动(1)" )
   END_RUNG wire#w1
   RUNG wire#w1
      Contact( "润滑故障分钟检测" )
      Coil( "润滑正常指示" )
   END_RUNG
   // the same network as SCL:
   #_w1 := "润滑电机启动" OR "润滑启动(1)";
   "润滑启动(1)" := #_w1 AND "润滑空开" AND "润滑电机停止" AND NOT "润滑故障";
   "润滑正常指示" := #_w1 AND "润滑故障分钟检测";
END_REGION

REGION Network 2
   RUNG wire#powerrail
      I_Contact( "润滑电机1过载" )
      wire#w1
      Contact( "故障复位" )
      Coil( "润滑电机过载" )
   END_RUNG
   RUNG wire#powerrail
      I_Contact( "润滑电机2过载_" )
   END_RUNG wire#w1
   RUNG wire#powerrail
      I_Contact( "润滑电机3过载_" )
   END_RUNG wire#w1
   RUNG wire#powerrail
      Contact( "润滑电机过载" )
   END_RUNG wire#w1
   // the same network as SCL:
   "润滑电机过载" := (NOT "润滑电机1过载" OR NOT "润滑电机2过载_" OR NOT "润滑电机3过载_" OR "润滑电机过载") AND "故障复位";
END_REGION

REGION Network 3
   RUNG wire#powerrail
      Contact( "润滑故障分钟检测" )
      wire#w1
      I_Contact( "低油压1" )
      wire#w2
      Contact( "故障复位" )
      Coil( "润滑油压低" )
   END_RUNG
   RUNG wire#w1
      I_Contact( "低油压2" )
   END_RUNG wire#w2
   RUNG wire#w1
      I_Contact( "低油压3" )
   END_RUNG wire#w2
   RUNG wire#w1
      Contact( "润滑油压低" )
   END_RUNG wire#w2
   // the same network as SCL:
   "润滑油压低" := "润滑故障分钟检测" AND (NOT "低油压1" OR NOT "低油压2" OR NOT "低油压3" OR "润滑油压低") AND "故障复位";
END_REGION

REGION Network 4
   RUNG wire#powerrail
      Contact( "润滑故障分钟检测" )
      wire#w1
      I_Contact( "高油压1" )
      wire#w2
      I_Contact( "故障复位" )
      Coil( "润滑高油压" )
   END_RUNG
   RUNG wire#w1
      I_Contact( "高油压2" )
   END_RUNG wire#w2
   RUNG wire#w1
      I_Contact( "高油压3" )
   END_RUNG wire#w2
   RUNG wire#w1
      Contact( "润滑高油压" )
   END_RUNG wire#w2
   // the same network as SCL:
   "润滑高油压" := "润滑故障分钟检测" AND (NOT "高油压1" OR NOT "高油压2" OR NOT "高油压3" OR "润滑高油压") AND NOT "故障复位";
END_REGION

REGION Network 5
   RUNG wire#powerrail
      Contact( "润滑故障分钟检测" )
      wire#w1
      Contact( "低油位" )
      wire#w2
      Contact( "故障复位" )
      Coil( "润滑低油位" )
   END_RUNG
   RUNG wire#w1
      Contact( "润滑低油位" )
   END_RUNG wire#w2
   // the same network as SCL:
   "润滑低油位" := "润滑故障分钟检测" AND ("低油位" OR "润滑低油位") AND "故障复位";
END_REGION

REGION Network 6
   RUNG wire#powerrail
      Contact( "润滑故障分钟检测" )
      wire#w1
      Contact( "高油位" )
      wire#w2
      Contact( "故障复位" )
      Coil( "油箱油位高指示" )
   END_RUNG
   RUNG wire#w1
      Contact( "油箱油位高指示" )
   END_RUNG wire#w2
   // the same network as SCL:
   "油箱油位高指示" := "润滑故障分钟检测" AND ("高油位" OR "油箱油位高指示") AND "故障复位";
END_REGION

REGION Network 7
   "计时器".润滑检测延时.TON(IN := "润滑启动(1)", PT := T#1M);
   "润滑故障分钟检测" := "计时器".润滑检测延时.Q;
END_REGION

REGION Network 8
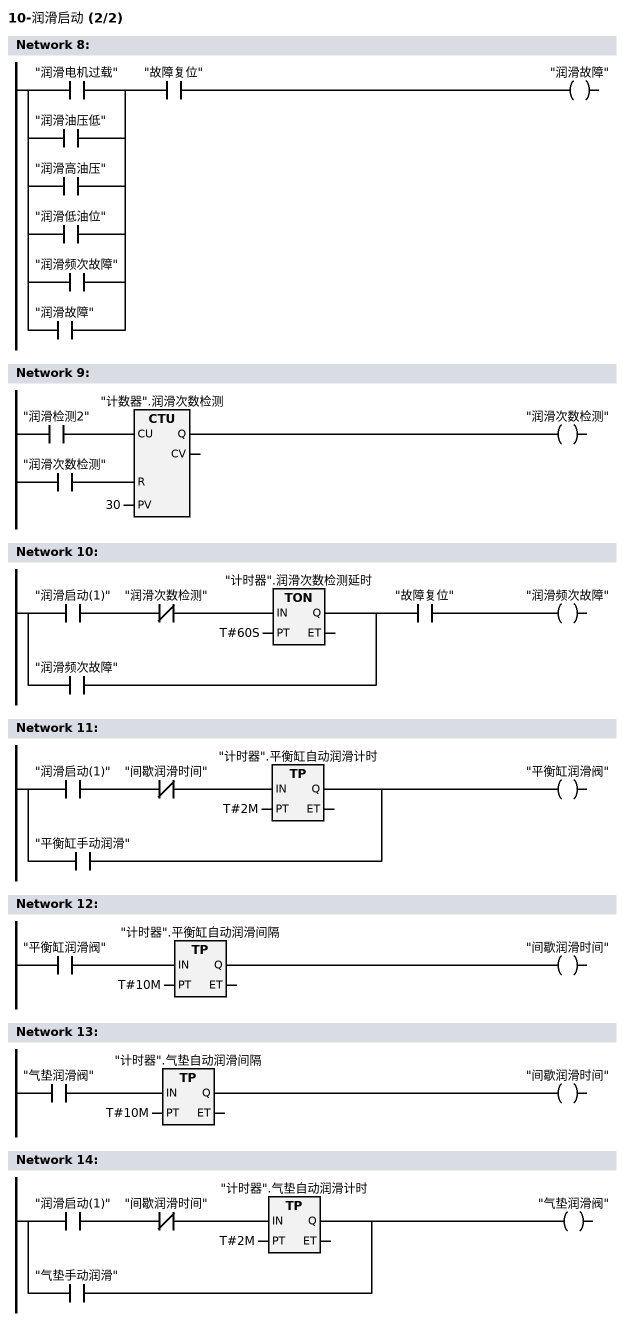
   RUNG wire#powerrail
      Contact( "润滑电机过载" )
      wire#w1
      Contact( "故障复位" )
      Coil( "润滑故障" )
   END_RUNG
   RUNG wire#powerrail
      Contact( "润滑油压低" )
   END_RUNG wire#w1
   RUNG wire#powerrail
      Contact( "润滑高油压" )
   END_RUNG wire#w1
   RUNG wire#powerrail
      Contact( "润滑低油位" )
   END_RUNG wire#w1
   RUNG wire#powerrail
      Contact( "润滑频次故障" )
   END_RUNG wire#w1
   RUNG wire#powerrail
      Contact( "润滑故障" )
   END_RUNG wire#w1
   // the same network as SCL:
   "润滑故障" := ("润滑电机过载" OR "润滑油压低" OR "润滑高油压" OR "润滑低油位" OR "润滑频次故障" OR "润滑故障") AND "故障复位";
END_REGION

REGION Network 9
   "计数器".润滑次数检测.CTU(CU := "润滑检测2", R := "润滑次数检测", PV := 30);
   "润滑次数检测" := "计数器".润滑次数检测.Q;
END_REGION

REGION Network 10
   "计时器".润滑次数检测延时.TON(IN := "润滑启动(1)" AND NOT "润滑次数检测", PT := T#60S);
   "润滑频次故障" := ("计时器".润滑次数检测延时.Q OR "润滑频次故障") AND "故障复位";
END_REGION

REGION Network 11
   "计时器".平衡缸自动润滑计时.TP(IN := "润滑启动(1)" AND NOT "间歇润滑时间", PT := T#2M);
   "平衡缸润滑阀" := "计时器".平衡缸自动润滑计时.Q OR "平衡缸手动润滑";
END_REGION

REGION Network 12
   "计时器".平衡缸自动润滑间隔.TP(IN := "平衡缸润滑阀", PT := T#10M);
   "间歇润滑时间" := "计时器".平衡缸自动润滑间隔.Q;
END_REGION

REGION Network 13
   "计时器".气垫自动润滑间隔.TP(IN := "气垫润滑阀", PT := T#10M);
   "间歇润滑时间" := "计时器".气垫自动润滑间隔.Q;
END_REGION

REGION Network 14
   "计时器".气垫自动润滑计时.TP(IN := "润滑启动(1)" AND NOT "间歇润滑时间", PT := T#2M);
   "气垫润滑阀" := "计时器".气垫自动润滑计时.Q OR "气垫手动润滑";
END_REGION
END_FUNCTION

FUNCTION "20-主电机启动程序" : Void   // FC20, LAD
{ S7_Optimized_Access := 'TRUE' }
VERSION : 0.1
BEGIN

REGION Network 1
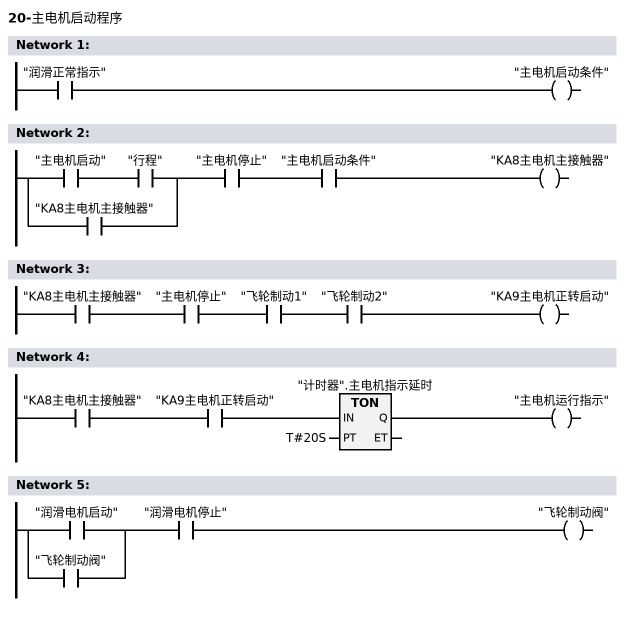
   RUNG wire#powerrail
      Contact( "润滑正常指示" )
      Coil( "主电机启动条件" )
   END_RUNG
   // the same network as SCL:
   "主电机启动条件" := "润滑正常指示";
END_REGION

REGION Network 2
   RUNG wire#powerrail
      Contact( "主电机启动" )
      Contact( "行程" )
      wire#w1
      Contact( "主电机停止" )
      Contact( "主电机启动条件" )
      Coil( "KA8主电机主接触器" )
   END_RUNG
   RUNG wire#powerrail
      Contact( "KA8主电机主接触器" )
   END_RUNG wire#w1
   // the same network as SCL:
   "KA8主电机主接触器" := (("主电机启动" AND "行程") OR "KA8主电机主接触器") AND "主电机停止" AND "主电机启动条件";
END_REGION

REGION Network 3
   RUNG wire#powerrail
      Contact( "KA8主电机主接触器" )
      Contact( "主电机停止" )
      Contact( "飞轮制动1" )
      Contact( "飞轮制动2" )
      Coil( "KA9主电机正转启动" )
   END_RUNG
   // the same network as SCL:
   "KA9主电机正转启动" := "KA8主电机主接触器" AND "主电机停止" AND "飞轮制动1" AND "飞轮制动2";
END_REGION

REGION Network 4
   "计时器".主电机指示延时.TON(IN := "KA8主电机主接触器" AND "KA9主电机正转启动", PT := T#20S);
   "主电机运行指示" := "计时器".主电机指示延时.Q;
END_REGION

REGION Network 5
   RUNG wire#powerrail
      Contact( "润滑电机启动" )
      wire#w1
      Contact( "润滑电机停止" )
      Coil( "飞轮制动阀" )
   END_RUNG
   RUNG wire#powerrail
      Contact( "飞轮制动阀" )
   END_RUNG wire#w1
   // the same network as SCL:
   "飞轮制动阀" := ("润滑电机启动" OR "飞轮制动阀") AND "润滑电机停止";
END_REGION
END_FUNCTION

FUNCTION "30-滑块行程" : Void   // FC30, LAD
{ S7_Optimized_Access := 'TRUE' }
VERSION : 0.1
   VAR_TEMP
      双手闭点检测 : Bool;
   END_VAR
BEGIN

REGION Network 1
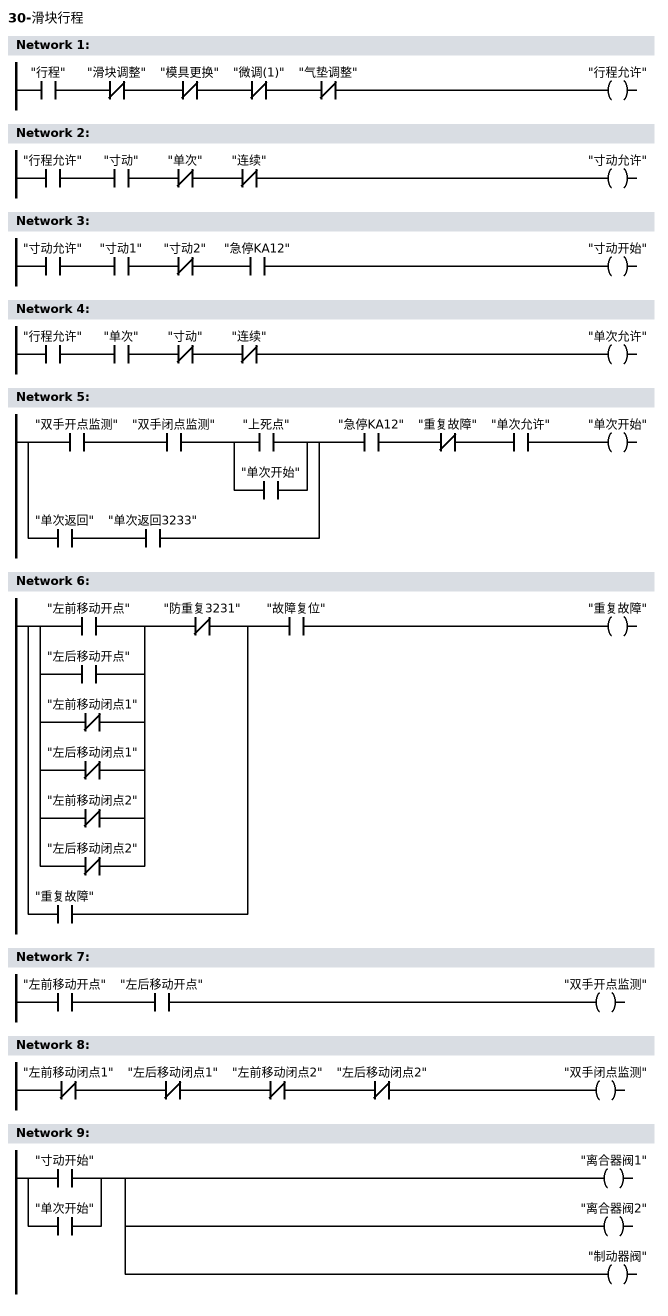
   RUNG wire#powerrail
      Contact( "行程" )
      I_Contact( "滑块调整" )
      I_Contact( "模具更换" )
      I_Contact( "微调(1)" )
      I_Contact( "气垫调整" )
      Coil( "行程允许" )
   END_RUNG
   // the same network as SCL:
   "行程允许" := "行程" AND NOT "滑块调整" AND NOT "模具更换" AND NOT "微调(1)" AND NOT "气垫调整";
END_REGION

REGION Network 2
   RUNG wire#powerrail
      Contact( "行程允许" )
      Contact( "寸动" )
      I_Contact( "单次" )
      I_Contact( "连续" )
      Coil( "寸动允许" )
   END_RUNG
   // the same network as SCL:
   "寸动允许" := "行程允许" AND "寸动" AND NOT "单次" AND NOT "连续";
END_REGION

REGION Network 3
   RUNG wire#powerrail
      Contact( "寸动允许" )
      Contact( "寸动1" )
      I_Contact( "寸动2" )
      Contact( "急停KA12" )
      Coil( "寸动开始" )
   END_RUNG
   // the same network as SCL:
   "寸动开始" := "寸动允许" AND "寸动1" AND NOT "寸动2" AND "急停KA12";
END_REGION

REGION Network 4
   RUNG wire#powerrail
      Contact( "行程允许" )
      Contact( "单次" )
      I_Contact( "寸动" )
      I_Contact( "连续" )
      Coil( "单次允许" )
   END_RUNG
   // the same network as SCL:
   "单次允许" := "行程允许" AND "单次" AND NOT "寸动" AND NOT "连续";
END_REGION

REGION Network 5
   RUNG wire#powerrail
      Contact( "双手开点监测" )
      Contact( "双手闭点监测" )
      wire#w1
      Contact( "上死点" )
      wire#w2
      Contact( "急停KA12" )
      I_Contact( "重复故障" )
      Contact( "单次允许" )
      Coil( "单次开始" )
   END_RUNG
   RUNG wire#w1
      Contact( "单次开始" )
   END_RUNG wire#w2
   RUNG wire#powerrail
      Contact( "单次返回" )
      Contact( "单次返回3233" )
   END_RUNG wire#w2
   // the same network as SCL:
   "单次开始" := (("双手开点监测" AND "双手闭点监测" AND ("上死点" OR "单次开始")) OR ("单次返回" AND "单次返回3233")) AND "急停KA12" AND NOT "重复故障" AND "单次允许";
END_REGION

REGION Network 6
   RUNG wire#powerrail
      Contact( "左前移动开点" )
      wire#w1
      I_Contact( "防重复3231" )
      wire#w2
      Contact( "故障复位" )
      Coil( "重复故障" )
   END_RUNG
   RUNG wire#powerrail
      Contact( "左后移动开点" )
   END_RUNG wire#w1
   RUNG wire#powerrail
      I_Contact( "左前移动闭点1" )
   END_RUNG wire#w1
   RUNG wire#powerrail
      I_Contact( "左后移动闭点1" )
   END_RUNG wire#w1
   RUNG wire#powerrail
      I_Contact( "左前移动闭点2" )
   END_RUNG wire#w1
   RUNG wire#powerrail
      I_Contact( "左后移动闭点2" )
   END_RUNG wire#w1
   RUNG wire#powerrail
      Contact( "重复故障" )
   END_RUNG wire#w2
   // the same network as SCL:
   "重复故障" := ((("左前移动开点" OR "左后移动开点" OR NOT "左前移动闭点1" OR NOT "左后移动闭点1" OR NOT "左前移动闭点2" OR NOT "左后移动闭点2") AND NOT "防重复3231") OR "重复故障") AND "故障复位";
END_REGION

REGION Network 7
   RUNG wire#powerrail
      Contact( "左前移动开点" )
      Contact( "左后移动开点" )
      Coil( "双手开点监测" )
   END_RUNG
   // the same network as SCL:
   "双手开点监测" := "左前移动开点" AND "左后移动开点";
END_REGION

REGION Network 8
   RUNG wire#powerrail
      I_Contact( "左前移动闭点1" )
      I_Contact( "左后移动闭点1" )
      I_Contact( "左前移动闭点2" )
      I_Contact( "左后移动闭点2" )
      Coil( "双手闭点监测" )
   END_RUNG
   // the same network as SCL:
   "双手闭点监测" := NOT "左前移动闭点1" AND NOT "左后移动闭点1" AND NOT "左前移动闭点2" AND NOT "左后移动闭点2";
END_REGION

REGION Network 9
   RUNG wire#powerrail
      Contact( "寸动开始" )
      wire#w1
      Coil( "离合器阀1" )
   END_RUNG
   RUNG wire#powerrail
      Contact( "单次开始" )
   END_RUNG wire#w1
   RUNG wire#w1
      Coil( "离合器阀2" )
   END_RUNG
   RUNG wire#w1
      Coil( "制动器阀" )
   END_RUNG
   // the same network as SCL:
   "离合器阀1" := "寸动开始" OR "单次开始";
   "离合器阀2" := "离合器阀1";
   "制动器阀" := "离合器阀1";
END_REGION
END_FUNCTION

FUNCTION "40-滑块调整程序" : Void   // FC40, LAD
{ S7_Optimized_Access := 'TRUE' }
VERSION : 0.1
BEGIN

REGION Network 1
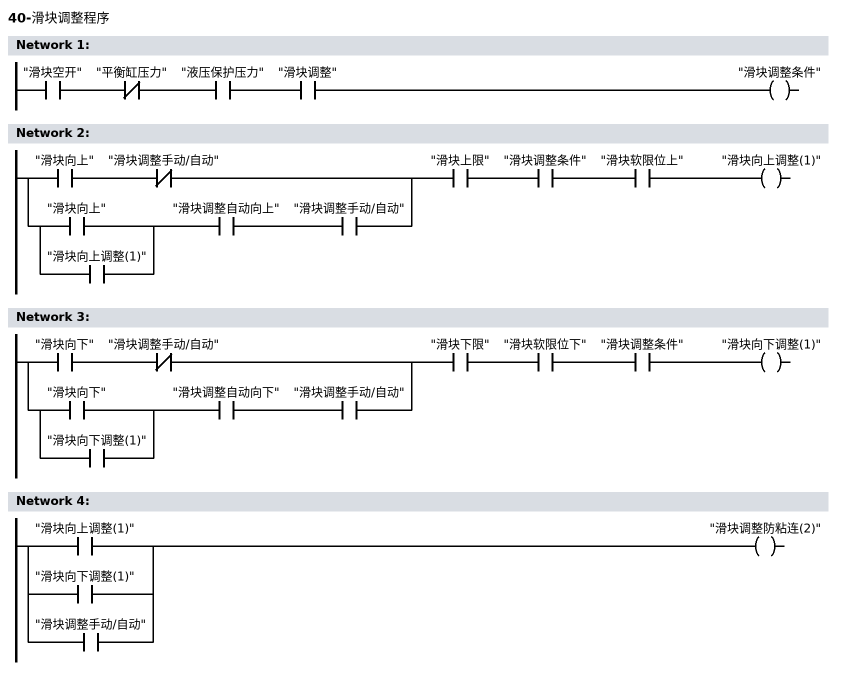
   RUNG wire#powerrail
      Contact( "滑块空开" )
      I_Contact( "平衡缸压力" )
      Contact( "液压保护压力" )
      Contact( "滑块调整" )
      Coil( "滑块调整条件" )
   END_RUNG
   // the same network as SCL:
   "滑块调整条件" := "滑块空开" AND NOT "平衡缸压力" AND "液压保护压力" AND "滑块调整";
END_REGION

REGION Network 2
   RUNG wire#powerrail
      Contact( "滑块向上" )
      I_Contact( "滑块调整手动/自动" )
      wire#w1
      Contact( "滑块上限" )
      Contact( "滑块调整条件" )
      Contact( "滑块软限位上" )
      Coil( "滑块向上调整(1)" )
   END_RUNG
   RUNG wire#powerrail
      Contact( "滑块向上" )
      wire#w2
      Contact( "滑块调整自动向上" )
      Contact( "滑块调整手动/自动" )
   END_RUNG wire#w1
   RUNG wire#powerrail
      Contact( "滑块向上调整(1)" )
   END_RUNG wire#w2
   // the same network as SCL:
   "滑块向上调整(1)" := (("滑块向上" AND NOT "滑块调整手动/自动") OR (("滑块向上" OR "滑块向上调整(1)") AND "滑块调整自动向上" AND "滑块调整手动/自动")) AND "滑块上限" AND "滑块调整条件" AND "滑块软限位上";
END_REGION

REGION Network 3
   RUNG wire#powerrail
      Contact( "滑块向下" )
      I_Contact( "滑块调整手动/自动" )
      wire#w1
      Contact( "滑块下限" )
      Contact( "滑块软限位下" )
      Contact( "滑块调整条件" )
      Coil( "滑块向下调整(1)" )
   END_RUNG
   RUNG wire#powerrail
      Contact( "滑块向下" )
      wire#w2
      Contact( "滑块调整自动向下" )
      Contact( "滑块调整手动/自动" )
   END_RUNG wire#w1
   RUNG wire#powerrail
      Contact( "滑块向下调整(1)" )
   END_RUNG wire#w2
   // the same network as SCL:
   "滑块向下调整(1)" := (("滑块向下" AND NOT "滑块调整手动/自动") OR (("滑块向下" OR "滑块向下调整(1)") AND "滑块调整自动向下" AND "滑块调整手动/自动")) AND "滑块下限" AND "滑块软限位下" AND "滑块调整条件";
END_REGION

REGION Network 4
   RUNG wire#powerrail
      Contact( "滑块向上调整(1)" )
      wire#w1
      Coil( "滑块调整防粘连(2)" )
   END_RUNG
   RUNG wire#powerrail
      Contact( "滑块向下调整(1)" )
   END_RUNG wire#w1
   RUNG wire#powerrail
      Contact( "滑块调整手动/自动" )
   END_RUNG wire#w1
   // the same network as SCL:
   "滑块调整防粘连(2)" := "滑块向上调整(1)" OR "滑块向下调整(1)" OR "滑块调整手动/自动";
END_REGION
END_FUNCTION

FUNCTION "50-移动工作台程序" : Void   // FC50, LAD
{ S7_Optimized_Access := 'TRUE' }
VERSION : 0.1
BEGIN

REGION Network 1
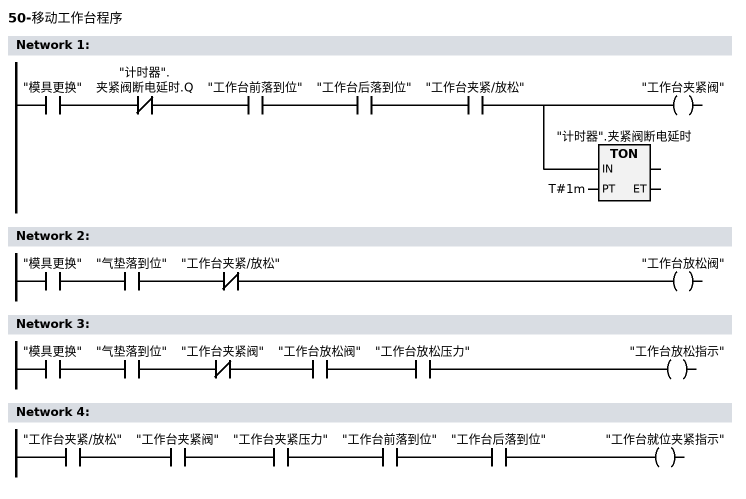
   "工作台夹紧阀" := "模具更换" AND NOT "计时器".夹紧阀断电延时.Q AND "工作台前落到位" AND "工作台后落到位" AND "工作台夹紧/放松";
   "计时器".夹紧阀断电延时.TON(IN := "工作台夹紧阀", PT := T#1m);
END_REGION

REGION Network 2
   RUNG wire#powerrail
      Contact( "模具更换" )
      Contact( "气垫落到位" )
      I_Contact( "工作台夹紧/放松" )
      Coil( "工作台放松阀" )
   END_RUNG
   // the same network as SCL:
   "工作台放松阀" := "模具更换" AND "气垫落到位" AND NOT "工作台夹紧/放松";
END_REGION

REGION Network 3
   RUNG wire#powerrail
      Contact( "模具更换" )
      Contact( "气垫落到位" )
      I_Contact( "工作台夹紧阀" )
      Contact( "工作台放松阀" )
      Contact( "工作台放松压力" )
      Coil( "工作台放松指示" )
   END_RUNG
   // the same network as SCL:
   "工作台放松指示" := "模具更换" AND "气垫落到位" AND NOT "工作台夹紧阀" AND "工作台放松阀" AND "工作台放松压力";
END_REGION

REGION Network 4
   RUNG wire#powerrail
      Contact( "工作台夹紧/放松" )
      Contact( "工作台夹紧阀" )
      Contact( "工作台夹紧压力" )
      Contact( "工作台前落到位" )
      Contact( "工作台后落到位" )
      Coil( "工作台就位夹紧指示" )
   END_RUNG
   // the same network as SCL:
   "工作台就位夹紧指示" := "工作台夹紧/放松" AND "工作台夹紧阀" AND "工作台夹紧压力" AND "工作台前落到位" AND "工作台后落到位";
END_REGION
END_FUNCTION

FUNCTION "60-气垫控制" : Void   // FC60, LAD
{ S7_Optimized_Access := 'TRUE' }
VERSION : 0.1
BEGIN

REGION Network 1
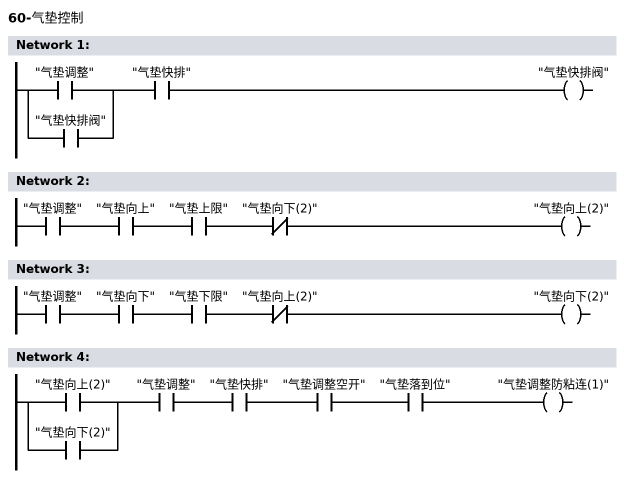
   RUNG wire#powerrail
      Contact( "气垫调整" )
      wire#w1
      Contact( "气垫快排" )
      Coil( "气垫快排阀" )
   END_RUNG
   RUNG wire#powerrail
      Contact( "气垫快排阀" )
   END_RUNG wire#w1
   // the same network as SCL:
   "气垫快排阀" := ("气垫调整" OR "气垫快排阀") AND "气垫快排";
END_REGION

REGION Network 2
   RUNG wire#powerrail
      Contact( "气垫调整" )
      Contact( "气垫向上" )
      Contact( "气垫上限" )
      I_Contact( "气垫向下(2)" )
      Coil( "气垫向上(2)" )
   END_RUNG
   // the same network as SCL:
   "气垫向上(2)" := "气垫调整" AND "气垫向上" AND "气垫上限" AND NOT "气垫向下(2)";
END_REGION

REGION Network 3
   RUNG wire#powerrail
      Contact( "气垫调整" )
      Contact( "气垫向下" )
      Contact( "气垫下限" )
      I_Contact( "气垫向上(2)" )
      Coil( "气垫向下(2)" )
   END_RUNG
   // the same network as SCL:
   "气垫向下(2)" := "气垫调整" AND "气垫向下" AND "气垫下限" AND NOT "气垫向上(2)";
END_REGION

REGION Network 4
   RUNG wire#powerrail
      Contact( "气垫向上(2)" )
      wire#w1
      Contact( "气垫调整" )
      Contact( "气垫快排" )
      Contact( "气垫调整空开" )
      Contact( "气垫落到位" )
      Coil( "气垫调整防粘连(1)" )
   END_RUNG
   RUNG wire#powerrail
      Contact( "气垫向下(2)" )
   END_RUNG wire#w1
   // the same network as SCL:
   "气垫调整防粘连(1)" := ("气垫向上(2)" OR "气垫向下(2)") AND "气垫调整" AND "气垫快排" AND "气垫调整空开" AND "气垫落到位";
END_REGION
END_FUNCTION

FUNCTION "70-液压保护" : Void   // FC70, LAD
{ S7_Optimized_Access := 'TRUE' }
VERSION : 0.1
BEGIN

REGION Network 1
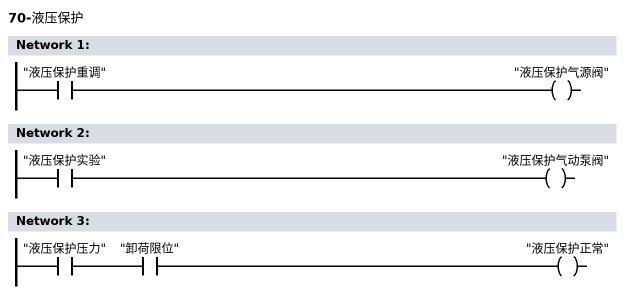
   RUNG wire#powerrail
      Contact( "液压保护重调" )
      Coil( "液压保护气源阀" )
   END_RUNG
   // the same network as SCL:
   "液压保护气源阀" := "液压保护重调";
END_REGION

REGION Network 2
   RUNG wire#powerrail
      Contact( "液压保护实验" )
      Coil( "液压保护气动泵阀" )
   END_RUNG
   // the same network as SCL:
   "液压保护气动泵阀" := "液压保护实验";
END_REGION

REGION Network 3
   RUNG wire#powerrail
      Contact( "液压保护压力" )
      Contact( "卸荷限位" )
      Coil( "液压保护正常" )
   END_RUNG
   // the same network as SCL:
   "液压保护正常" := "液压保护压力" AND "卸荷限位";
END_REGION
END_FUNCTION

FUNCTION "80-产品计数" : Void   // FC80, LAD
{ S7_Optimized_Access := 'TRUE' }
VERSION : 0.1
BEGIN

REGION Network 1
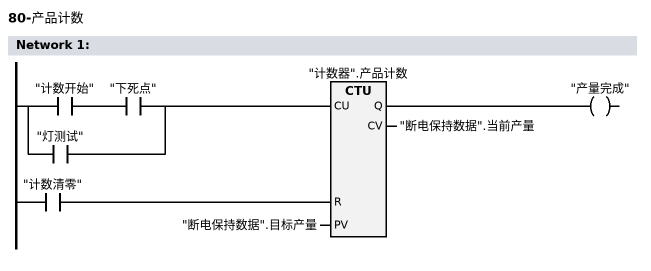
   "计数器".产品计数.CTU(CU := ("计数开始" AND "下死点") OR "灯测试", R := "计数清零", PV := "断电保持数据".目标产量, CV => "断电保持数据".当前产量);
   "产量完成" := "计数器".产品计数.Q;
END_REGION
END_FUNCTION

FUNCTION "横梁编码器调制" : Void   // FC90, LAD
{ S7_Optimized_Access := 'TRUE' }
VERSION : 0.1
BEGIN

REGION Network 1
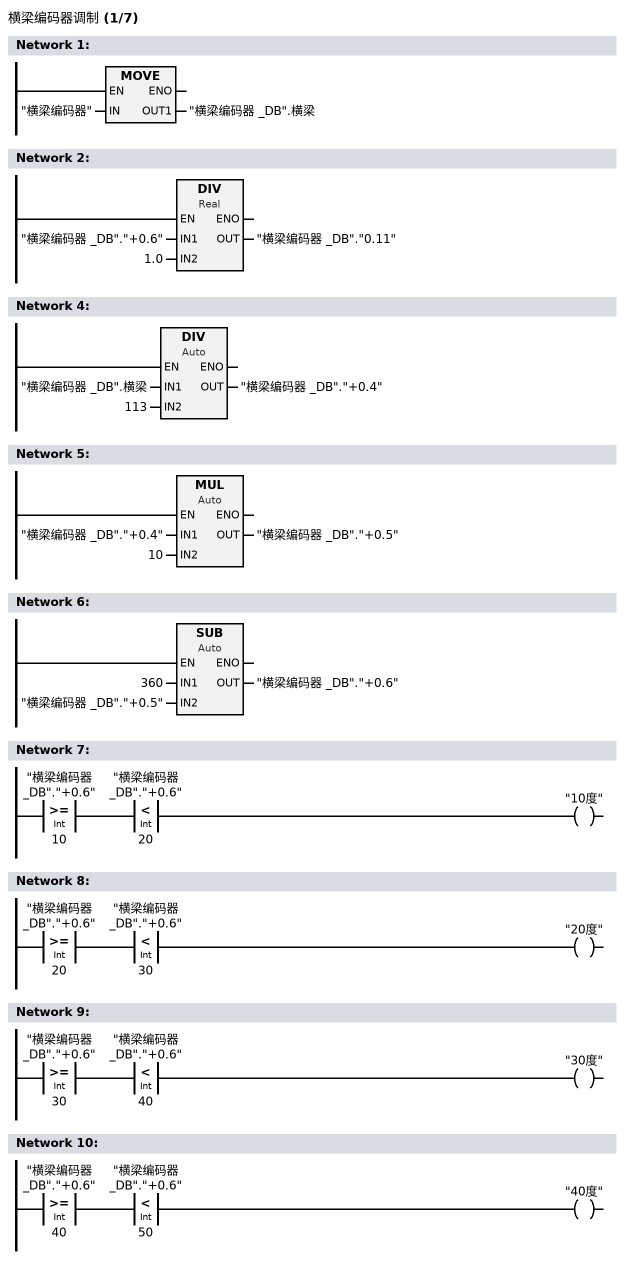
   RUNG wire#powerrail
      Move(in := "横梁编码器", out1 => "横梁编码器 _DB".横梁)
   END_RUNG
   // the same network as SCL:
   "横梁编码器 _DB".横梁 := "横梁编码器";
END_REGION

REGION Network 2
   RUNG wire#powerrail
      { S7_Templates := "SrcType := Real" } Div(in1 := "横梁编码器 _DB"."+0.6", in2 := 1.0, out => "横梁编码器 _DB"."0.11")
   END_RUNG
   // the same network as SCL:
   "横梁编码器 _DB"."0.11" := "横梁编码器 _DB"."+0.6" / 1.0;
END_REGION

REGION Network 4
   RUNG wire#powerrail
      Div(in1 := "横梁编码器 _DB".横梁, in2 := 113, out => "横梁编码器 _DB"."+0.4")
   END_RUNG
   // the same network as SCL:
   "横梁编码器 _DB"."+0.4" := "横梁编码器 _DB".横梁 / 113;
END_REGION

REGION Network 5
   RUNG wire#powerrail
      Mul(in1 := "横梁编码器 _DB"."+0.4", in2 := 10, out => "横梁编码器 _DB"."+0.5")
   END_RUNG
   // the same network as SCL:
   "横梁编码器 _DB"."+0.5" := "横梁编码器 _DB"."+0.4" * 10;
END_REGION

REGION Network 6
   RUNG wire#powerrail
      Sub(in1 := 360, in2 := "横梁编码器 _DB"."+0.5", out => "横梁编码器 _DB"."+0.6")
   END_RUNG
   // the same network as SCL:
   "横梁编码器 _DB"."+0.6" := 360 - "横梁编码器 _DB"."+0.5";
END_REGION

REGION Network 7
   RUNG wire#powerrail
      { S7_Templates := "SrcType := Int" } GE_Contact(in1 := "横梁编码器 _DB"."+0.6", in2 := 10)
      { S7_Templates := "SrcType := Int" } LT_Contact(in1 := "横梁编码器 _DB"."+0.6", in2 := 20)
      Coil( "10度" )
   END_RUNG
   // the same network as SCL:
   "10度" := ("横梁编码器 _DB"."+0.6" >= 10) AND ("横梁编码器 _DB"."+0.6" < 20);
END_REGION

REGION Network 8
   RUNG wire#powerrail
      { S7_Templates := "SrcType := Int" } GE_Contact(in1 := "横梁编码器 _DB"."+0.6", in2 := 20)
      { S7_Templates := "SrcType := Int" } LT_Contact(in1 := "横梁编码器 _DB"."+0.6", in2 := 30)
      Coil( "20度" )
   END_RUNG
   // the same network as SCL:
   "20度" := ("横梁编码器 _DB"."+0.6" >= 20) AND ("横梁编码器 _DB"."+0.6" < 30);
END_REGION

REGION Network 9
   RUNG wire#powerrail
      { S7_Templates := "SrcType := Int" } GE_Contact(in1 := "横梁编码器 _DB"."+0.6", in2 := 30)
      { S7_Templates := "SrcType := Int" } LT_Contact(in1 := "横梁编码器 _DB"."+0.6", in2 := 40)
      Coil( "30度" )
   END_RUNG
   // the same network as SCL:
   "30度" := ("横梁编码器 _DB"."+0.6" >= 30) AND ("横梁编码器 _DB"."+0.6" < 40);
END_REGION

REGION Network 10
   RUNG wire#powerrail
      { S7_Templates := "SrcType := Int" } GE_Contact(in1 := "横梁编码器 _DB"."+0.6", in2 := 40)
      { S7_Templates := "SrcType := Int" } LT_Contact(in1 := "横梁编码器 _DB"."+0.6", in2 := 50)
      Coil( "40度" )
   END_RUNG
   // the same network as SCL:
   "40度" := ("横梁编码器 _DB"."+0.6" >= 40) AND ("横梁编码器 _DB"."+0.6" < 50);
END_REGION

REGION Network 11
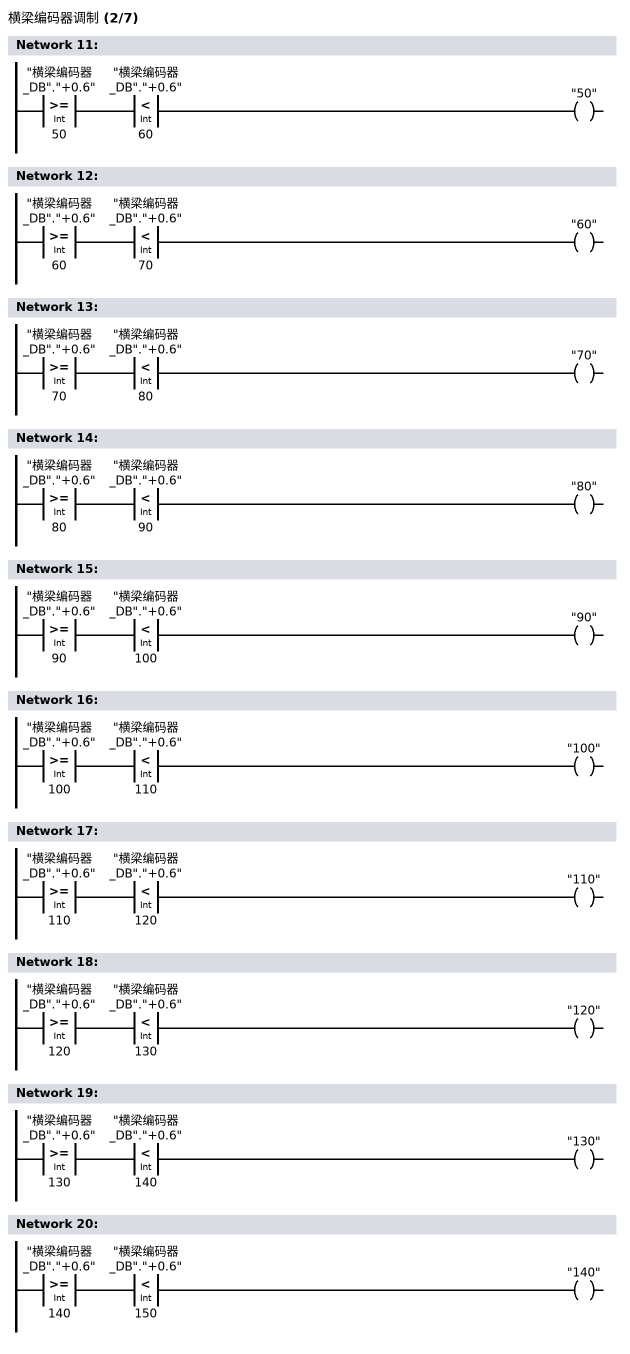
   RUNG wire#powerrail
      { S7_Templates := "SrcType := Int" } GE_Contact(in1 := "横梁编码器 _DB"."+0.6", in2 := 50)
      { S7_Templates := "SrcType := Int" } LT_Contact(in1 := "横梁编码器 _DB"."+0.6", in2 := 60)
      Coil( "50" )
   END_RUNG
   // the same network as SCL:
   "50" := ("横梁编码器 _DB"."+0.6" >= 50) AND ("横梁编码器 _DB"."+0.6" < 60);
END_REGION

REGION Network 12
   RUNG wire#powerrail
      { S7_Templates := "SrcType := Int" } GE_Contact(in1 := "横梁编码器 _DB"."+0.6", in2 := 60)
      { S7_Templates := "SrcType := Int" } LT_Contact(in1 := "横梁编码器 _DB"."+0.6", in2 := 70)
      Coil( "60" )
   END_RUNG
   // the same network as SCL:
   "60" := ("横梁编码器 _DB"."+0.6" >= 60) AND ("横梁编码器 _DB"."+0.6" < 70);
END_REGION

REGION Network 13
   RUNG wire#powerrail
      { S7_Templates := "SrcType := Int" } GE_Contact(in1 := "横梁编码器 _DB"."+0.6", in2 := 70)
      { S7_Templates := "SrcType := Int" } LT_Contact(in1 := "横梁编码器 _DB"."+0.6", in2 := 80)
      Coil( "70" )
   END_RUNG
   // the same network as SCL:
   "70" := ("横梁编码器 _DB"."+0.6" >= 70) AND ("横梁编码器 _DB"."+0.6" < 80);
END_REGION

REGION Network 14
   RUNG wire#powerrail
      { S7_Templates := "SrcType := Int" } GE_Contact(in1 := "横梁编码器 _DB"."+0.6", in2 := 80)
      { S7_Templates := "SrcType := Int" } LT_Contact(in1 := "横梁编码器 _DB"."+0.6", in2 := 90)
      Coil( "80" )
   END_RUNG
   // the same network as SCL:
   "80" := ("横梁编码器 _DB"."+0.6" >= 80) AND ("横梁编码器 _DB"."+0.6" < 90);
END_REGION

REGION Network 15
   RUNG wire#powerrail
      { S7_Templates := "SrcType := Int" } GE_Contact(in1 := "横梁编码器 _DB"."+0.6", in2 := 90)
      { S7_Templates := "SrcType := Int" } LT_Contact(in1 := "横梁编码器 _DB"."+0.6", in2 := 100)
      Coil( "90" )
   END_RUNG
   // the same network as SCL:
   "90" := ("横梁编码器 _DB"."+0.6" >= 90) AND ("横梁编码器 _DB"."+0.6" < 100);
END_REGION

REGION Network 16
   RUNG wire#powerrail
      { S7_Templates := "SrcType := Int" } GE_Contact(in1 := "横梁编码器 _DB"."+0.6", in2 := 100)
      { S7_Templates := "SrcType := Int" } LT_Contact(in1 := "横梁编码器 _DB"."+0.6", in2 := 110)
      Coil( "100" )
   END_RUNG
   // the same network as SCL:
   "100" := ("横梁编码器 _DB"."+0.6" >= 100) AND ("横梁编码器 _DB"."+0.6" < 110);
END_REGION

REGION Network 17
   RUNG wire#powerrail
      { S7_Templates := "SrcType := Int" } GE_Contact(in1 := "横梁编码器 _DB"."+0.6", in2 := 110)
      { S7_Templates := "SrcType := Int" } LT_Contact(in1 := "横梁编码器 _DB"."+0.6", in2 := 120)
      Coil( "110" )
   END_RUNG
   // the same network as SCL:
   "110" := ("横梁编码器 _DB"."+0.6" >= 110) AND ("横梁编码器 _DB"."+0.6" < 120);
END_REGION

REGION Network 18
   RUNG wire#powerrail
      { S7_Templates := "SrcType := Int" } GE_Contact(in1 := "横梁编码器 _DB"."+0.6", in2 := 120)
      { S7_Templates := "SrcType := Int" } LT_Contact(in1 := "横梁编码器 _DB"."+0.6", in2 := 130)
      Coil( "120" )
   END_RUNG
   // the same network as SCL:
   "120" := ("横梁编码器 _DB"."+0.6" >= 120) AND ("横梁编码器 _DB"."+0.6" < 130);
END_REGION

REGION Network 19
   RUNG wire#powerrail
      { S7_Templates := "SrcType := Int" } GE_Contact(in1 := "横梁编码器 _DB"."+0.6", in2 := 130)
      { S7_Templates := "SrcType := Int" } LT_Contact(in1 := "横梁编码器 _DB"."+0.6", in2 := 140)
      Coil( "130" )
   END_RUNG
   // the same network as SCL:
   "130" := ("横梁编码器 _DB"."+0.6" >= 130) AND ("横梁编码器 _DB"."+0.6" < 140);
END_REGION

REGION Network 20
   RUNG wire#powerrail
      { S7_Templates := "SrcType := Int" } GE_Contact(in1 := "横梁编码器 _DB"."+0.6", in2 := 140)
      { S7_Templates := "SrcType := Int" } LT_Contact(in1 := "横梁编码器 _DB"."+0.6", in2 := 150)
      Coil( "140" )
   END_RUNG
   // the same network as SCL:
   "140" := ("横梁编码器 _DB"."+0.6" >= 140) AND ("横梁编码器 _DB"."+0.6" < 150);
END_REGION

REGION Network 21
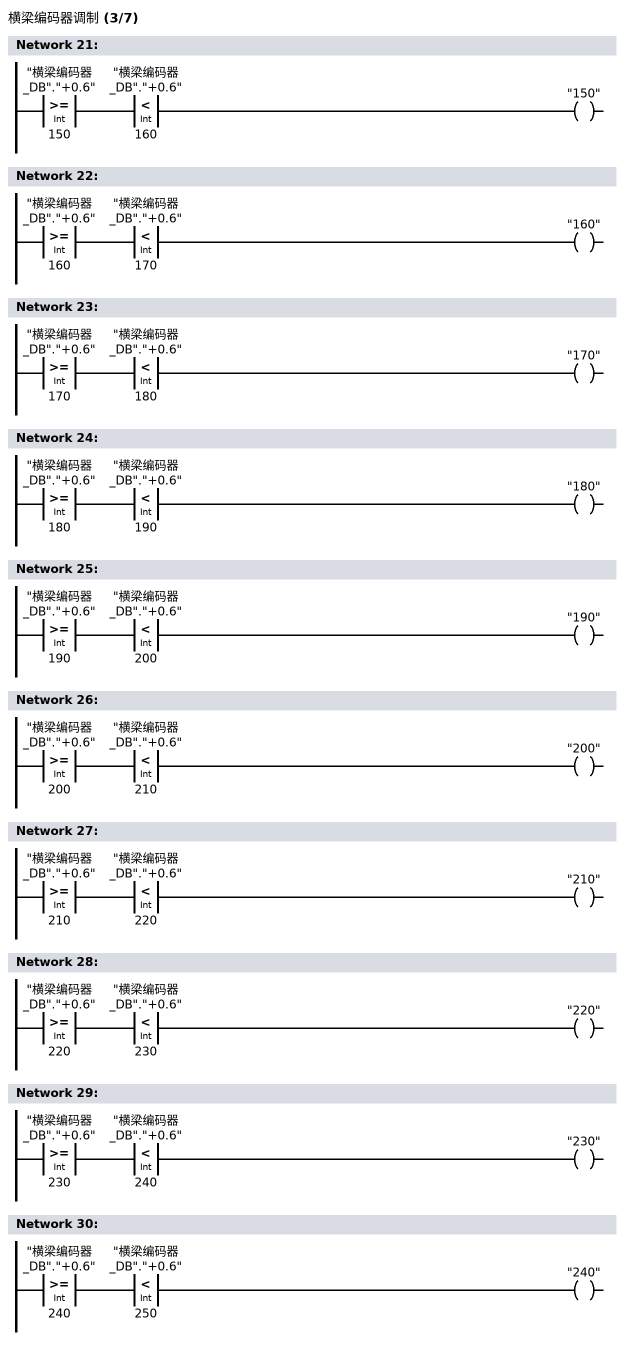
   RUNG wire#powerrail
      { S7_Templates := "SrcType := Int" } GE_Contact(in1 := "横梁编码器 _DB"."+0.6", in2 := 150)
      { S7_Templates := "SrcType := Int" } LT_Contact(in1 := "横梁编码器 _DB"."+0.6", in2 := 160)
      Coil( "150" )
   END_RUNG
   // the same network as SCL:
   "150" := ("横梁编码器 _DB"."+0.6" >= 150) AND ("横梁编码器 _DB"."+0.6" < 160);
END_REGION

REGION Network 22
   RUNG wire#powerrail
      { S7_Templates := "SrcType := Int" } GE_Contact(in1 := "横梁编码器 _DB"."+0.6", in2 := 160)
      { S7_Templates := "SrcType := Int" } LT_Contact(in1 := "横梁编码器 _DB"."+0.6", in2 := 170)
      Coil( "160" )
   END_RUNG
   // the same network as SCL:
   "160" := ("横梁编码器 _DB"."+0.6" >= 160) AND ("横梁编码器 _DB"."+0.6" < 170);
END_REGION

REGION Network 23
   RUNG wire#powerrail
      { S7_Templates := "SrcType := Int" } GE_Contact(in1 := "横梁编码器 _DB"."+0.6", in2 := 170)
      { S7_Templates := "SrcType := Int" } LT_Contact(in1 := "横梁编码器 _DB"."+0.6", in2 := 180)
      Coil( "170" )
   END_RUNG
   // the same network as SCL:
   "170" := ("横梁编码器 _DB"."+0.6" >= 170) AND ("横梁编码器 _DB"."+0.6" < 180);
END_REGION

REGION Network 24
   RUNG wire#powerrail
      { S7_Templates := "SrcType := Int" } GE_Contact(in1 := "横梁编码器 _DB"."+0.6", in2 := 180)
      { S7_Templates := "SrcType := Int" } LT_Contact(in1 := "横梁编码器 _DB"."+0.6", in2 := 190)
      Coil( "180" )
   END_RUNG
   // the same network as SCL:
   "180" := ("横梁编码器 _DB"."+0.6" >= 180) AND ("横梁编码器 _DB"."+0.6" < 190);
END_REGION

REGION Network 25
   RUNG wire#powerrail
      { S7_Templates := "SrcType := Int" } GE_Contact(in1 := "横梁编码器 _DB"."+0.6", in2 := 190)
      { S7_Templates := "SrcType := Int" } LT_Contact(in1 := "横梁编码器 _DB"."+0.6", in2 := 200)
      Coil( "190" )
   END_RUNG
   // the same network as SCL:
   "190" := ("横梁编码器 _DB"."+0.6" >= 190) AND ("横梁编码器 _DB"."+0.6" < 200);
END_REGION

REGION Network 26
   RUNG wire#powerrail
      { S7_Templates := "SrcType := Int" } GE_Contact(in1 := "横梁编码器 _DB"."+0.6", in2 := 200)
      { S7_Templates := "SrcType := Int" } LT_Contact(in1 := "横梁编码器 _DB"."+0.6", in2 := 210)
      Coil( "200" )
   END_RUNG
   // the same network as SCL:
   "200" := ("横梁编码器 _DB"."+0.6" >= 200) AND ("横梁编码器 _DB"."+0.6" < 210);
END_REGION

REGION Network 27
   RUNG wire#powerrail
      { S7_Templates := "SrcType := Int" } GE_Contact(in1 := "横梁编码器 _DB"."+0.6", in2 := 210)
      { S7_Templates := "SrcType := Int" } LT_Contact(in1 := "横梁编码器 _DB"."+0.6", in2 := 220)
      Coil( "210" )
   END_RUNG
   // the same network as SCL:
   "210" := ("横梁编码器 _DB"."+0.6" >= 210) AND ("横梁编码器 _DB"."+0.6" < 220);
END_REGION

REGION Network 28
   RUNG wire#powerrail
      { S7_Templates := "SrcType := Int" } GE_Contact(in1 := "横梁编码器 _DB"."+0.6", in2 := 220)
      { S7_Templates := "SrcType := Int" } LT_Contact(in1 := "横梁编码器 _DB"."+0.6", in2 := 230)
      Coil( "220" )
   END_RUNG
   // the same network as SCL:
   "220" := ("横梁编码器 _DB"."+0.6" >= 220) AND ("横梁编码器 _DB"."+0.6" < 230);
END_REGION

REGION Network 29
   RUNG wire#powerrail
      { S7_Templates := "SrcType := Int" } GE_Contact(in1 := "横梁编码器 _DB"."+0.6", in2 := 230)
      { S7_Templates := "SrcType := Int" } LT_Contact(in1 := "横梁编码器 _DB"."+0.6", in2 := 240)
      Coil( "230" )
   END_RUNG
   // the same network as SCL:
   "230" := ("横梁编码器 _DB"."+0.6" >= 230) AND ("横梁编码器 _DB"."+0.6" < 240);
END_REGION

REGION Network 30
   RUNG wire#powerrail
      { S7_Templates := "SrcType := Int" } GE_Contact(in1 := "横梁编码器 _DB"."+0.6", in2 := 240)
      { S7_Templates := "SrcType := Int" } LT_Contact(in1 := "横梁编码器 _DB"."+0.6", in2 := 250)
      Coil( "240" )
   END_RUNG
   // the same network as SCL:
   "240" := ("横梁编码器 _DB"."+0.6" >= 240) AND ("横梁编码器 _DB"."+0.6" < 250);
END_REGION

REGION Network 31
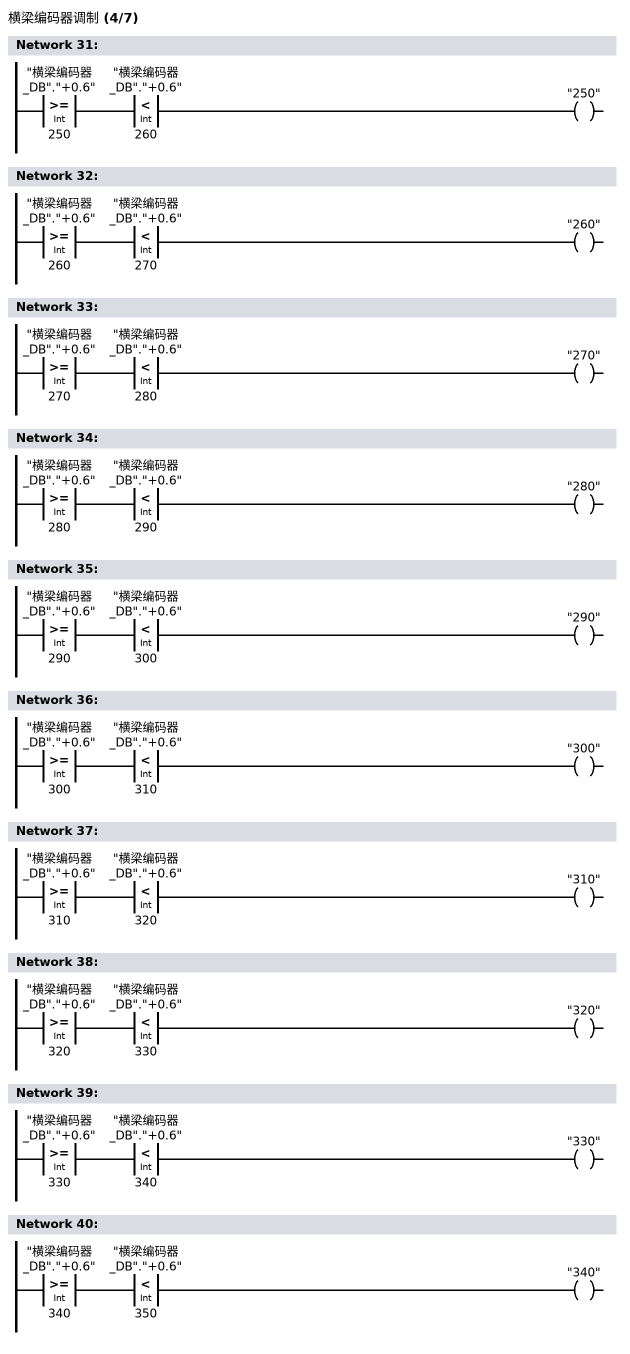
   RUNG wire#powerrail
      { S7_Templates := "SrcType := Int" } GE_Contact(in1 := "横梁编码器 _DB"."+0.6", in2 := 250)
      { S7_Templates := "SrcType := Int" } LT_Contact(in1 := "横梁编码器 _DB"."+0.6", in2 := 260)
      Coil( "250" )
   END_RUNG
   // the same network as SCL:
   "250" := ("横梁编码器 _DB"."+0.6" >= 250) AND ("横梁编码器 _DB"."+0.6" < 260);
END_REGION

REGION Network 32
   RUNG wire#powerrail
      { S7_Templates := "SrcType := Int" } GE_Contact(in1 := "横梁编码器 _DB"."+0.6", in2 := 260)
      { S7_Templates := "SrcType := Int" } LT_Contact(in1 := "横梁编码器 _DB"."+0.6", in2 := 270)
      Coil( "260" )
   END_RUNG
   // the same network as SCL:
   "260" := ("横梁编码器 _DB"."+0.6" >= 260) AND ("横梁编码器 _DB"."+0.6" < 270);
END_REGION

REGION Network 33
   RUNG wire#powerrail
      { S7_Templates := "SrcType := Int" } GE_Contact(in1 := "横梁编码器 _DB"."+0.6", in2 := 270)
      { S7_Templates := "SrcType := Int" } LT_Contact(in1 := "横梁编码器 _DB"."+0.6", in2 := 280)
      Coil( "270" )
   END_RUNG
   // the same network as SCL:
   "270" := ("横梁编码器 _DB"."+0.6" >= 270) AND ("横梁编码器 _DB"."+0.6" < 280);
END_REGION

REGION Network 34
   RUNG wire#powerrail
      { S7_Templates := "SrcType := Int" } GE_Contact(in1 := "横梁编码器 _DB"."+0.6", in2 := 280)
      { S7_Templates := "SrcType := Int" } LT_Contact(in1 := "横梁编码器 _DB"."+0.6", in2 := 290)
      Coil( "280" )
   END_RUNG
   // the same network as SCL:
   "280" := ("横梁编码器 _DB"."+0.6" >= 280) AND ("横梁编码器 _DB"."+0.6" < 290);
END_REGION

REGION Network 35
   RUNG wire#powerrail
      { S7_Templates := "SrcType := Int" } GE_Contact(in1 := "横梁编码器 _DB"."+0.6", in2 := 290)
      { S7_Templates := "SrcType := Int" } LT_Contact(in1 := "横梁编码器 _DB"."+0.6", in2 := 300)
      Coil( "290" )
   END_RUNG
   // the same network as SCL:
   "290" := ("横梁编码器 _DB"."+0.6" >= 290) AND ("横梁编码器 _DB"."+0.6" < 300);
END_REGION

REGION Network 36
   RUNG wire#powerrail
      { S7_Templates := "SrcType := Int" } GE_Contact(in1 := "横梁编码器 _DB"."+0.6", in2 := 300)
      { S7_Templates := "SrcType := Int" } LT_Contact(in1 := "横梁编码器 _DB"."+0.6", in2 := 310)
      Coil( "300" )
   END_RUNG
   // the same network as SCL:
   "300" := ("横梁编码器 _DB"."+0.6" >= 300) AND ("横梁编码器 _DB"."+0.6" < 310);
END_REGION

REGION Network 37
   RUNG wire#powerrail
      { S7_Templates := "SrcType := Int" } GE_Contact(in1 := "横梁编码器 _DB"."+0.6", in2 := 310)
      { S7_Templates := "SrcType := Int" } LT_Contact(in1 := "横梁编码器 _DB"."+0.6", in2 := 320)
      Coil( "310" )
   END_RUNG
   // the same network as SCL:
   "310" := ("横梁编码器 _DB"."+0.6" >= 310) AND ("横梁编码器 _DB"."+0.6" < 320);
END_REGION

REGION Network 38
   RUNG wire#powerrail
      { S7_Templates := "SrcType := Int" } GE_Contact(in1 := "横梁编码器 _DB"."+0.6", in2 := 320)
      { S7_Templates := "SrcType := Int" } LT_Contact(in1 := "横梁编码器 _DB"."+0.6", in2 := 330)
      Coil( "320" )
   END_RUNG
   // the same network as SCL:
   "320" := ("横梁编码器 _DB"."+0.6" >= 320) AND ("横梁编码器 _DB"."+0.6" < 330);
END_REGION

REGION Network 39
   RUNG wire#powerrail
      { S7_Templates := "SrcType := Int" } GE_Contact(in1 := "横梁编码器 _DB"."+0.6", in2 := 330)
      { S7_Templates := "SrcType := Int" } LT_Contact(in1 := "横梁编码器 _DB"."+0.6", in2 := 340)
      Coil( "330" )
   END_RUNG
   // the same network as SCL:
   "330" := ("横梁编码器 _DB"."+0.6" >= 330) AND ("横梁编码器 _DB"."+0.6" < 340);
END_REGION

REGION Network 40
   RUNG wire#powerrail
      { S7_Templates := "SrcType := Int" } GE_Contact(in1 := "横梁编码器 _DB"."+0.6", in2 := 340)
      { S7_Templates := "SrcType := Int" } LT_Contact(in1 := "横梁编码器 _DB"."+0.6", in2 := 350)
      Coil( "340" )
   END_RUNG
   // the same network as SCL:
   "340" := ("横梁编码器 _DB"."+0.6" >= 340) AND ("横梁编码器 _DB"."+0.6" < 350);
END_REGION

REGION Network 41
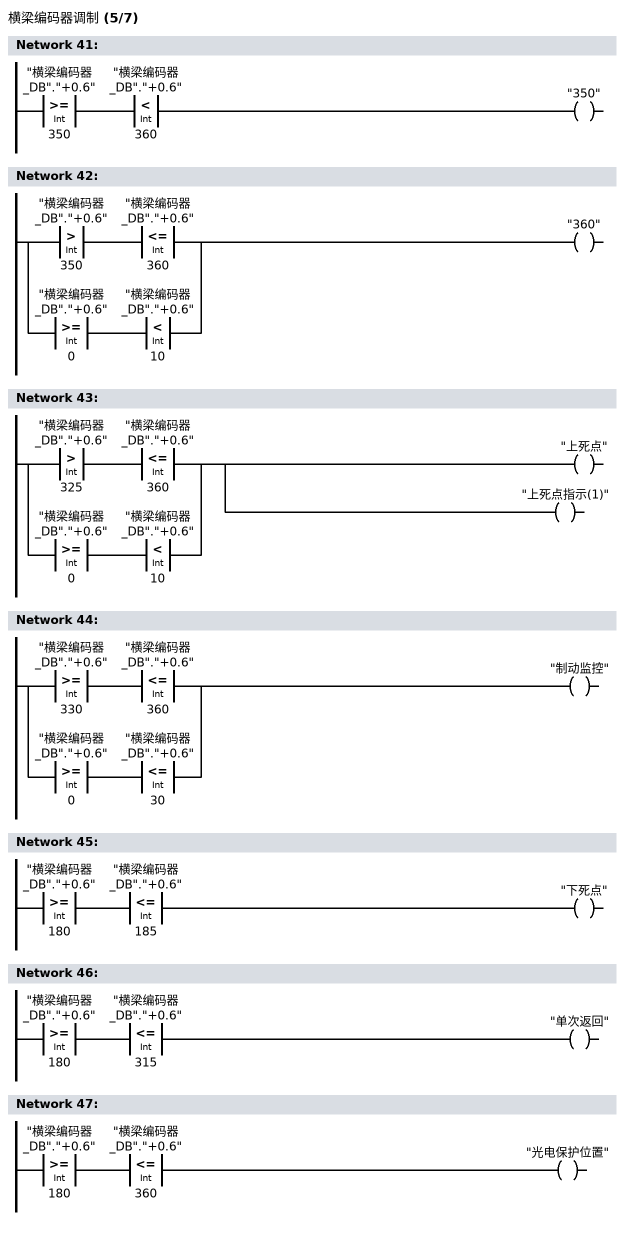
   RUNG wire#powerrail
      { S7_Templates := "SrcType := Int" } GE_Contact(in1 := "横梁编码器 _DB"."+0.6", in2 := 350)
      { S7_Templates := "SrcType := Int" } LT_Contact(in1 := "横梁编码器 _DB"."+0.6", in2 := 360)
      Coil( "350" )
   END_RUNG
   // the same network as SCL:
   "350" := ("横梁编码器 _DB"."+0.6" >= 350) AND ("横梁编码器 _DB"."+0.6" < 360);
END_REGION

REGION Network 42
   RUNG wire#powerrail
      { S7_Templates := "SrcType := Int" } GT_Contact(in1 := "横梁编码器 _DB"."+0.6", in2 := 350)
      { S7_Templates := "SrcType := Int" } LE_Contact(in1 := "横梁编码器 _DB"."+0.6", in2 := 360)
      wire#w1
      Coil( "360" )
   END_RUNG
   RUNG wire#powerrail
      { S7_Templates := "SrcType := Int" } GE_Contact(in1 := "横梁编码器 _DB"."+0.6", in2 := 0)
      { S7_Templates := "SrcType := Int" } LT_Contact(in1 := "横梁编码器 _DB"."+0.6", in2 := 10)
   END_RUNG wire#w1
   // the same network as SCL:
   "360" := (("横梁编码器 _DB"."+0.6" > 350) AND ("横梁编码器 _DB"."+0.6" <= 360)) OR (("横梁编码器 _DB"."+0.6" >= 0) AND ("横梁编码器 _DB"."+0.6" < 10));
END_REGION

REGION Network 43
   RUNG wire#powerrail
      { S7_Templates := "SrcType := Int" } GT_Contact(in1 := "横梁编码器 _DB"."+0.6", in2 := 325)
      { S7_Templates := "SrcType := Int" } LE_Contact(in1 := "横梁编码器 _DB"."+0.6", in2 := 360)
      wire#w1
      Coil( "上死点" )
   END_RUNG
   RUNG wire#powerrail
      { S7_Templates := "SrcType := Int" } GE_Contact(in1 := "横梁编码器 _DB"."+0.6", in2 := 0)
      { S7_Templates := "SrcType := Int" } LT_Contact(in1 := "横梁编码器 _DB"."+0.6", in2 := 10)
   END_RUNG wire#w1
   RUNG wire#w1
      Coil( "上死点指示(1)" )
   END_RUNG
   // the same network as SCL:
   "上死点" := (("横梁编码器 _DB"."+0.6" > 325) AND ("横梁编码器 _DB"."+0.6" <= 360)) OR (("横梁编码器 _DB"."+0.6" >= 0) AND ("横梁编码器 _DB"."+0.6" < 10));
   "上死点指示(1)" := "上死点";
END_REGION

REGION Network 44
   RUNG wire#powerrail
      { S7_Templates := "SrcType := Int" } GE_Contact(in1 := "横梁编码器 _DB"."+0.6", in2 := 330)
      { S7_Templates := "SrcType := Int" } LE_Contact(in1 := "横梁编码器 _DB"."+0.6", in2 := 360)
      wire#w1
      Coil( "制动监控" )
   END_RUNG
   RUNG wire#powerrail
      { S7_Templates := "SrcType := Int" } GE_Contact(in1 := "横梁编码器 _DB"."+0.6", in2 := 0)
      { S7_Templates := "SrcType := Int" } LE_Contact(in1 := "横梁编码器 _DB"."+0.6", in2 := 30)
   END_RUNG wire#w1
   // the same network as SCL:
   "制动监控" := (("横梁编码器 _DB"."+0.6" >= 330) AND ("横梁编码器 _DB"."+0.6" <= 360)) OR (("横梁编码器 _DB"."+0.6" >= 0) AND ("横梁编码器 _DB"."+0.6" <= 30));
END_REGION

REGION Network 45
   RUNG wire#powerrail
      { S7_Templates := "SrcType := Int" } GE_Contact(in1 := "横梁编码器 _DB"."+0.6", in2 := 180)
      { S7_Templates := "SrcType := Int" } LE_Contact(in1 := "横梁编码器 _DB"."+0.6", in2 := 185)
      Coil( "下死点" )
   END_RUNG
   // the same network as SCL:
   "下死点" := ("横梁编码器 _DB"."+0.6" >= 180) AND ("横梁编码器 _DB"."+0.6" <= 185);
END_REGION

REGION Network 46
   RUNG wire#powerrail
      { S7_Templates := "SrcType := Int" } GE_Contact(in1 := "横梁编码器 _DB"."+0.6", in2 := 180)
      { S7_Templates := "SrcType := Int" } LE_Contact(in1 := "横梁编码器 _DB"."+0.6", in2 := 315)
      Coil( "单次返回" )
   END_RUNG
   // the same network as SCL:
   "单次返回" := ("横梁编码器 _DB"."+0.6" >= 180) AND ("横梁编码器 _DB"."+0.6" <= 315);
END_REGION

REGION Network 47
   RUNG wire#powerrail
      { S7_Templates := "SrcType := Int" } GE_Contact(in1 := "横梁编码器 _DB"."+0.6", in2 := 180)
      { S7_Templates := "SrcType := Int" } LE_Contact(in1 := "横梁编码器 _DB"."+0.6", in2 := 360)
      Coil( "光电保护位置" )
   END_RUNG
   // the same network as SCL:
   "光电保护位置" := ("横梁编码器 _DB"."+0.6" >= 180) AND ("横梁编码器 _DB"."+0.6" <= 360);
END_REGION

REGION Network 48
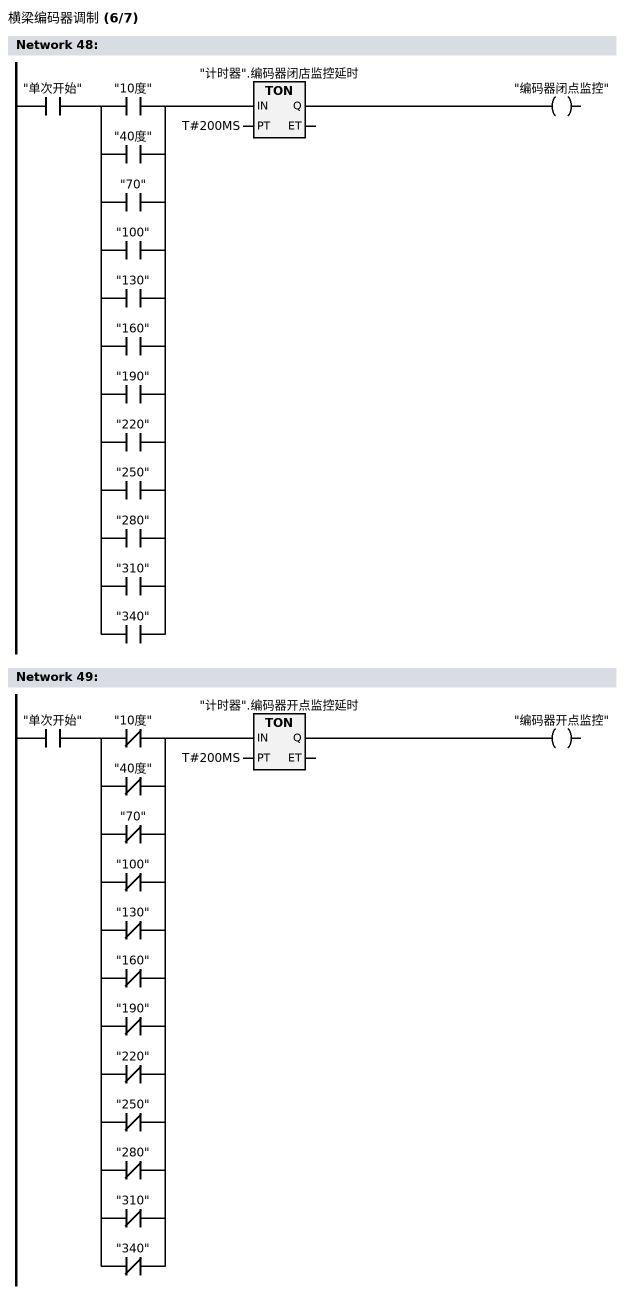
   "计时器".编码器闭店监控延时.TON(IN := "单次开始" AND ("10度" OR "40度" OR "70" OR "100" OR "130" OR "160" OR "190" OR "220" OR "250" OR "280" OR "310" OR "340"),
                       PT := T#200MS);
   "编码器闭点监控" := "计时器".编码器闭店监控延时.Q;
END_REGION

REGION Network 49
   "计时器".编码器开点监控延时.TON(IN := "单次开始" AND (NOT "10度" OR NOT "40度" OR NOT "70" OR NOT "100" OR NOT "130" OR NOT "160" OR NOT "190" OR NOT "220" OR NOT "250" OR NOT "280" OR NOT "310" OR NOT "340"),
                       PT := T#200MS);
   "编码器开点监控" := "计时器".编码器开点监控延时.Q;
END_REGION

REGION Network 50
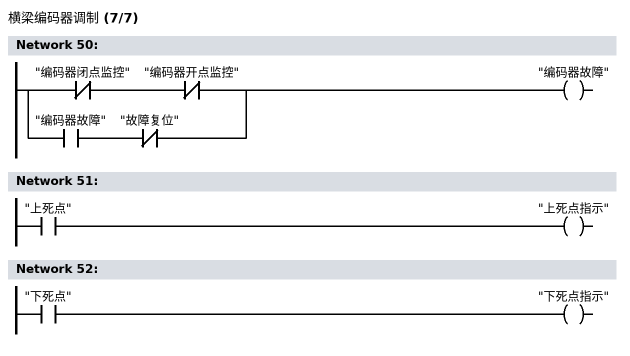
   RUNG wire#powerrail
      I_Contact( "编码器闭点监控" )
      I_Contact( "编码器开点监控" )
      wire#w1
      Coil( "编码器故障" )
   END_RUNG
   RUNG wire#powerrail
      Contact( "编码器故障" )
      I_Contact( "故障复位" )
   END_RUNG wire#w1
   // the same network as SCL:
   "编码器故障" := (NOT "编码器闭点监控" AND NOT "编码器开点监控") OR ("编码器故障" AND NOT "故障复位");
END_REGION

REGION Network 51
   RUNG wire#powerrail
      Contact( "上死点" )
      Coil( "上死点指示" )
   END_RUNG
   // the same network as SCL:
   "上死点指示" := "上死点";
END_REGION

REGION Network 52
   RUNG wire#powerrail
      Contact( "下死点" )
      Coil( "下死点指示" )
   END_RUNG
   // the same network as SCL:
   "下死点指示" := "下死点";
END_REGION
END_FUNCTION

FUNCTION "滑块编码器调制" : Void   // FC100, LAD
{ S7_Optimized_Access := 'TRUE' }
VERSION : 0.1
// 滑块编码器
   VAR_TEMP
      D102 : Real;
      D103 : Real;
   END_VAR
BEGIN

REGION Network 1
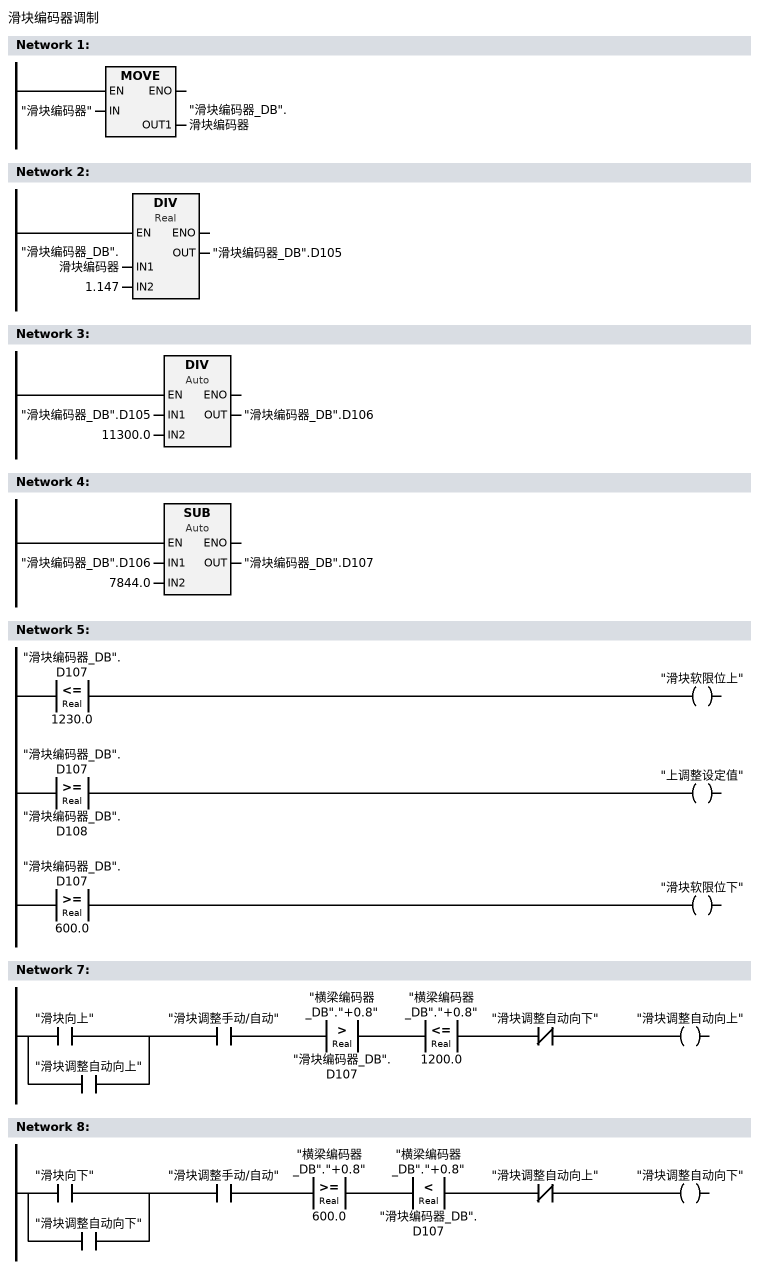
   RUNG wire#powerrail
      Move(in := "滑块编码器", out1 => "滑块编码器_DB".滑块编码器)
   END_RUNG
   // the same network as SCL:
   "滑块编码器_DB".滑块编码器 := "滑块编码器";
END_REGION

REGION Network 2
   RUNG wire#powerrail
      { S7_Templates := "SrcType := Real" } Div(in1 := "滑块编码器_DB".滑块编码器, in2 := 1.147, out => "滑块编码器_DB".D105)
   END_RUNG
   // the same network as SCL:
   "滑块编码器_DB".D105 := "滑块编码器_DB".滑块编码器 / 1.147;
END_REGION

REGION Network 3
   RUNG wire#powerrail
      Div(in1 := "滑块编码器_DB".D105, in2 := 11300.0, out => "滑块编码器_DB".D106)
   END_RUNG
   // the same network as SCL:
   "滑块编码器_DB".D106 := "滑块编码器_DB".D105 / 11300.0;
END_REGION

REGION Network 4
   RUNG wire#powerrail
      Sub(in1 := "滑块编码器_DB".D106, in2 := 7844.0, out => "滑块编码器_DB".D107)
   END_RUNG
   // the same network as SCL:
   "滑块编码器_DB".D107 := "滑块编码器_DB".D106 - 7844.0;
END_REGION

REGION Network 5
   RUNG wire#powerrail
      { S7_Templates := "SrcType := Real" } LE_Contact(in1 := "滑块编码器_DB".D107, in2 := 1230.0)
      Coil( "滑块软限位上" )
   END_RUNG
   RUNG wire#powerrail
      { S7_Templates := "SrcType := Real" } GE_Contact(in1 := "滑块编码器_DB".D107, in2 := "滑块编码器_DB".D108)
      Coil( "上调整设定值" )
   END_RUNG
   RUNG wire#powerrail
      { S7_Templates := "SrcType := Real" } GE_Contact(in1 := "滑块编码器_DB".D107, in2 := 600.0)
      Coil( "滑块软限位下" )
   END_RUNG
   // the same network as SCL:
   "滑块软限位上" := "滑块编码器_DB".D107 <= 1230.0;
   "上调整设定值" := "滑块编码器_DB".D107 >= "滑块编码器_DB".D108;
   "滑块软限位下" := "滑块编码器_DB".D107 >= 600.0;
END_REGION

REGION Network 7
   RUNG wire#powerrail
      Contact( "滑块向上" )
      wire#w1
      Contact( "滑块调整手动/自动" )
      { S7_Templates := "SrcType := Real" } GT_Contact(in1 := "横梁编码器 _DB"."+0.8", in2 := "滑块编码器_DB".D107)
      { S7_Templates := "SrcType := Real" } LE_Contact(in1 := "横梁编码器 _DB"."+0.8", in2 := 1200.0)
      I_Contact( "滑块调整自动向下" )
      Coil( "滑块调整自动向上" )
   END_RUNG
   RUNG wire#powerrail
      Contact( "滑块调整自动向上" )
   END_RUNG wire#w1
   // the same network as SCL:
   "滑块调整自动向上" := ("滑块向上" OR "滑块调整自动向上") AND "滑块调整手动/自动" AND ("横梁编码器 _DB"."+0.8" > "滑块编码器_DB".D107) AND ("横梁编码器 _DB"."+0.8" <= 1200.0) AND NOT "滑块调整自动向下";
END_REGION

REGION Network 8
   RUNG wire#powerrail
      Contact( "滑块向下" )
      wire#w1
      Contact( "滑块调整手动/自动" )
      { S7_Templates := "SrcType := Real" } GE_Contact(in1 := "横梁编码器 _DB"."+0.8", in2 := 600.0)
      { S7_Templates := "SrcType := Real" } LT_Contact(in1 := "横梁编码器 _DB"."+0.8", in2 := "滑块编码器_DB".D107)
      I_Contact( "滑块调整自动向上" )
      Coil( "滑块调整自动向下" )
   END_RUNG
   RUNG wire#powerrail
      Contact( "滑块调整自动向下" )
   END_RUNG wire#w1
   // the same network as SCL:
   "滑块调整自动向下" := ("滑块向下" OR "滑块调整自动向下") AND "滑块调整手动/自动" AND ("横梁编码器 _DB"."+0.8" >= 600.0) AND ("横梁编码器 _DB"."+0.8" < "滑块编码器_DB".D107) AND NOT "滑块调整自动向上";
END_REGION
END_FUNCTION

ORGANIZATION_BLOCK "Main"   // OB1, LAD, ProgramCycle
TITLE = "Main Program Sweep (Cycle)"
{ S7_Optimized_Access := 'TRUE' }
VERSION : 0.1
   VAR_INPUT
      Initial_Call : Bool;   // Initial call of this OB
      Remanence : Bool;   // =True, if remanent data are available
   END_VAR
BEGIN

REGION Network 1
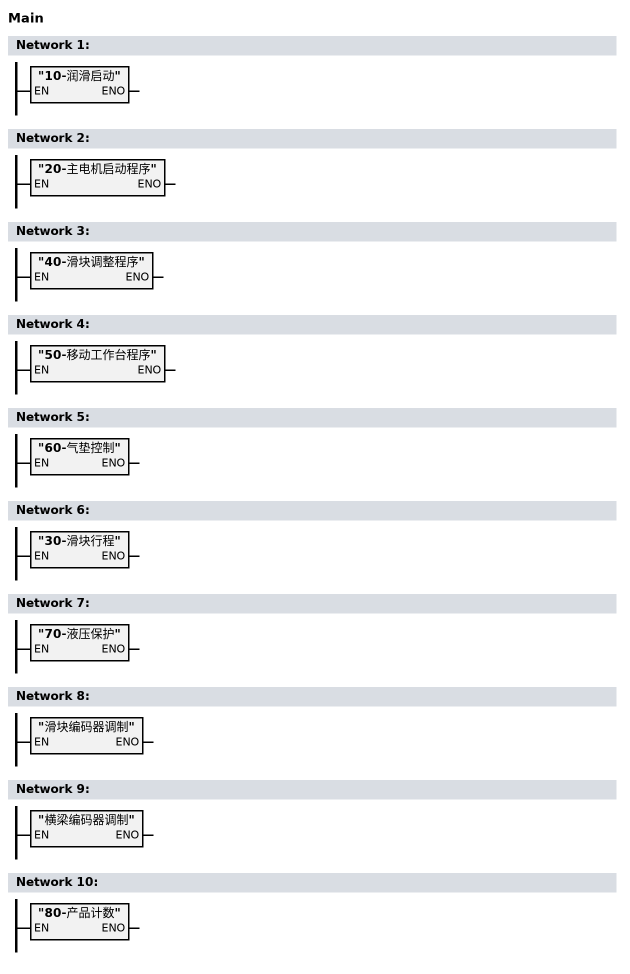
   RUNG wire#powerrail
      "10-润滑启动"()
   END_RUNG
   // the same network as SCL:
   "10-润滑启动"();
END_REGION

REGION Network 2
   RUNG wire#powerrail
      "20-主电机启动程序"()
   END_RUNG
   // the same network as SCL:
   "20-主电机启动程序"();
END_REGION

REGION Network 3
   RUNG wire#powerrail
      "40-滑块调整程序"()
   END_RUNG
   // the same network as SCL:
   "40-滑块调整程序"();
END_REGION

REGION Network 4
   RUNG wire#powerrail
      "50-移动工作台程序"()
   END_RUNG
   // the same network as SCL:
   "50-移动工作台程序"();
END_REGION

REGION Network 5
   RUNG wire#powerrail
      "60-气垫控制"()
   END_RUNG
   // the same network as SCL:
   "60-气垫控制"();
END_REGION

REGION Network 6
   RUNG wire#powerrail
      "30-滑块行程"()
   END_RUNG
   // the same network as SCL:
   "30-滑块行程"();
END_REGION

REGION Network 7
   RUNG wire#powerrail
      "70-液压保护"()
   END_RUNG
   // the same network as SCL:
   "70-液压保护"();
END_REGION

REGION Network 8
   RUNG wire#powerrail
      "滑块编码器调制"()
   END_RUNG
   // the same network as SCL:
   "滑块编码器调制"();
END_REGION

REGION Network 9
   RUNG wire#powerrail
      "横梁编码器调制"()
   END_RUNG
   // the same network as SCL:
   "横梁编码器调制"();
END_REGION

REGION Network 10
   RUNG wire#powerrail
      "80-产品计数"()
   END_RUNG
   // the same network as SCL:
   "80-产品计数"();
END_REGION
END_ORGANIZATION_BLOCK

ORGANIZATION_BLOCK "IO测试"   // OB125, LAD, ProgramCycle
TITLE = "Main Program Sweep (Cycle)"
{ S7_Optimized_Access := 'TRUE' }
VERSION : 0.1
   VAR_INPUT
      Initial_Call : Bool;   // Initial call of this OB
      Remanence : Bool;   // =True, if remanent data are available
   END_VAR
BEGIN
END_ORGANIZATION_BLOCK

(* ===== HMI "HMI_RT_1" =====
system functions are stored by id; their names below are inferred from use
connection "HMI_连接_1": ETHERNET, S7_1200_OMS

HMI tags "默认变量表"
   "主电机运行指示" : Bool = PLC 主电机运行指示 AT %Q10.5, 1 s
   "滑块向上" : Bool = PLC 滑块向上 AT %I13.0, 1 s
   "滑块向下KM7" : Bool = PLC "滑块向下调整(1)" AT %Q3.7, 1 s
   "滑块向上KM6" : Bool = PLC "滑块向上调整(1)" AT %Q3.6, 1 s
   "360" : Bool = PLC 360 AT %M204.3, 100 ms
   "10度" : Bool = PLC 10度 AT %M200.0, 100 ms
   "20度" : Bool = PLC 20度 AT %M200.1, 100 ms
   "30度" : Bool = PLC 30度 AT %M200.2, 100 ms
   "40度" : Bool = PLC 40度 AT %M200.3, 100 ms
   "50" : Bool = PLC 50 AT %M200.4, 100 ms
   "60" : Bool = PLC 60 AT %M200.5, 100 ms
   "70" : Bool = PLC 70 AT %M200.6, 100 ms
   "80" : Bool = PLC 80 AT %M200.7, 100 ms
   "90" : Bool = PLC 90 AT %M201.0, 100 ms
   "100" : Bool = PLC 100 AT %M201.1, 100 ms
   "110" : Bool = PLC 110 AT %M201.2, 100 ms
   "120" : Bool = PLC 120 AT %M201.3, 100 ms
   "130" : Bool = PLC 130 AT %M201.4, 100 ms
   "140" : Bool, internal
   "150" : Bool = PLC 150 AT %M201.6, 100 ms
   "160" : Bool = PLC 160 AT %M201.7, 100 ms
   "170" : Bool = PLC 170 AT %M202.0, 100 ms
   "180" : Bool = PLC 180 AT %M202.1, 100 ms
   "190" : Bool = PLC 190 AT %M202.2, 100 ms
   "200" : Bool = PLC 200 AT %M202.3, 100 ms
   "210" : Bool = PLC 210 AT %M202.4, 100 ms
   "220" : Bool = PLC 220 AT %M202.5, 100 ms
   "230" : Bool = PLC 230 AT %M202.6, 100 ms
   "240" : Bool = PLC 240 AT %M202.7, 100 ms
   "250" : Bool = PLC 250 AT %M203.0, 100 ms
   "260" : Bool = PLC 260 AT %M203.1, 100 ms
   "270" : Bool = PLC 270 AT %M203.2, 100 ms
   "280" : Bool = PLC 280 AT %M203.3, 100 ms
   "290" : Bool = PLC 290 AT %M203.4, 100 ms
   "300" : Bool = PLC 300 AT %M203.5, 100 ms
   "310" : Bool = PLC 310 AT %M203.6, 100 ms
   "320" : Bool = PLC 320 AT %M203.7, 100 ms
   "330" : Bool = PLC 330 AT %M204.0, 100 ms
   "340" : Bool = PLC 340 AT %M204.1, 100 ms
   "350" : Bool = PLC 350 AT %M204.2, 100 ms
   "工作台落到位前" : Bool = PLC 工作台前落到位 AT %I26.2, 1 s
   "工作台落到位后" : Bool = PLC 工作台后落到位 AT %I26.3, 1 s
   "工作台夹紧压检" : Bool = PLC 工作台夹紧压力 AT %I25.2, 1 s
   "工作台夹紧阀(1)" : Bool = PLC 工作台夹紧阀 AT %Q13.0, 1 s
   "平衡缸气压检测" : Bool = PLC 平衡缸压力 AT %I25.1, 1 s
   "润滑油泵启动OK" : Bool = PLC 润滑正常指示 AT %Q10.2, 1 s
   "润滑油压正常" : Bool = PLC 润滑正常指示 AT %Q10.2, 1 s
   "滤油器堵塞指示" : Bool = PLC 滤油器堵塞指示 AT %Q10.3, 1 s
   "急停开点左后" : Bool = PLC 设备故障指示 AT %Q11.2, 1 s
   "急停开点左前" : Bool = PLC 急停KA12 AT %I2.5, 1 s
   "爬梯开关" : Bool = PLC 梯子开关 AT %I18.1, 1 s
   "液压保护压力检测" : Bool = PLC 液压保护压力 AT %I22.4, 1 s
   "液压保护卸荷" : Bool = PLC 液压保护气源阀 AT %Q12.5, 1 s
   "液压保护故障" : Bool = PLC 液压保护正常指示 AT %Q10.6, 1 s
   "横梁编码器" : DWord = PLC 横梁编码器 AT %ID68, 1 s
   "ECamdata _DB_+0.7" : DInt = PLC 滑块编码器 AT %ID72, 1 s
   "横梁编码器 _DB_+0.6" : Int = PLC "横梁编码器 _DB"."+0.6", 1 s
   "上死点指示" : Bool = PLC 上死点指示 AT %M0.0, 1 s
   "工作台松开" : Bool = PLC "工作台夹紧/放松" AT %I13.4, 1 s
   "工作台放松阀(1)" : Bool = PLC 工作台放松阀 AT %Q13.1, 1 s
   "工作台放松压检" : Bool = PLC 工作台放松压力 AT %I25.3, 1 s
   "工作台落到位" : Bool = PLC 工作台就位夹紧指示 AT %Q11.5, 1 s
   "工作台夹紧" : Bool = PLC 工作台夹紧 AT %I24.6, 1 s
   "工作台-夹紧OK" : Bool = PLC 工作台就位夹紧指示 AT %Q11.5, 1 s
   "工作台放松OK" : Bool = PLC 工作台放松指示 AT %Q11.6, 1 s
   "横梁编码器 _DB_0.11" : Real = PLC "横梁编码器 _DB"."0.11", 1 s
   "滑块调整自动选择" : Bool = PLC 滑块调整自动选择 AT %M16.2, 1 s
   "ECamdata _DB_+0.36" : Int = PLC 滑块编码器_DB."+0.36", 100 ms
   "ECamdata _DB_+0.47" : Real = PLC 滑块编码器_DB."+0.47", 100 ms
   "ECamdata _DB_+0.6" : Int = PLC 滑块编码器_DB.电子凸轮编码器显示, 100 ms
   "ECamdata _DB_AQD" : Real = PLC 滑块编码器_DB.平衡器压力显示, 100 ms
   "ECamdata _DB_AQD2" : Real = PLC 滑块编码器_DB.AQD2, 100 ms
   "ECamdata _DB_AQD3" : Real = PLC 滑块编码器_DB.气垫模拟量显示1, 100 ms
   "ECamdata _DB_D{0}" : Real = PLC 滑块编码器_DB.D[0], 100 ms
   "ECamdata _DB_D{1}" : Real = PLC 滑块编码器_DB.D[1], 100 ms
   "ECamdata _DB_D{10}滑块设定高度" : Real = PLC 滑块编码器_DB.D[10], 100 ms
   "ECamdata _DB_D{11}" : Real = PLC 滑块编码器_DB.D[11], 100 ms
   "ECamdata _DB_D{6}" : Real = PLC 滑块编码器_DB.D[6], 100 ms
   "ECamdata _DB_D{7}" : Real = PLC 滑块编码器_DB.D[7], 100 ms
   "ECamdata _DB_D{9}" : Real = PLC 滑块编码器_DB.D[9], 100 ms
   "ECamdata _DB_D102" : Int = PLC 滑块编码器_DB.D102, 100 ms
   "ECamdata _DB_D107" : Int = PLC 滑块编码器_DB.D107, 1 s
   "ECamdata _DB_D108" : Real = PLC 滑块编码器_DB.D108, 1 s
   "ECamdata _DB_当前产量" : Int = PLC 滑块编码器_DB.当前产量, 1 s
   "ECamdata _DB_滑块打油次数" : Int = PLC 滑块编码器_DB.滑块打油次数, 100 ms
   "ECamdata _DB_平衡器设置压力" : Real = PLC 滑块编码器_DB.平衡器设置压力, 100 ms
   "ECamdata _DB_气垫2压力设置" : Real = PLC 滑块编码器_DB.气垫2压力设置, 100 ms
   "ECamdata _DB_气垫模拟量显示1" : Real = PLC 滑块编码器_DB.气垫模拟量显示2, 100 ms
   "ECamdata _DB_气垫压力设置" : Real = PLC 滑块编码器_DB.气垫1压力设置, 100 ms
   "ECamdata _DB_设置产量" : Int = PLC 滑块编码器_DB.设置产量, 1 s
   "ECamdata _DB_主分油器打油次数" : Int = PLC 滑块编码器_DB.主分油器打油次数, 100 ms
   "滑块调整手动/自动" : Bool = PLC "滑块调整手动/自动" AT %I13.2, 100 ms
   "横梁编码器 _DB_+0.8" : Int = PLC "横梁编码器 _DB"."+0.8", 1 s
   "PLC报警变量组1" : Bool = PLC 设备故障指示 AT %Q11.2, 1 s
   "PLC报警变量组2" : Bool = PLC 梯子开关 AT %I18.1, 1 s
   "气垫落到位" : Bool = PLC 气垫落到位 AT %I24.4, 1 s
   "工作台落到位后(1)" : Bool = PLC 工作台前落到位 AT %I26.2, 1 s
   "横梁编码器 _DB_+0.6(1)" : Int = PLC "横梁编码器 _DB"."+0.6" AT %DB1.DBX0.0, 1 s
   "上死点" : Bool = PLC 上死点 AT %M204.4, 1 s
   "气垫上限" : Bool = PLC 气垫上限 AT %I23.4, 1 s
   "气垫下限" : Bool = PLC 气垫下限 AT %I23.5, 1 s
   "气垫调整空开" : Bool = PLC 气垫调整空开 AT %I3.6, 1 s
   "气垫调整" : Bool = PLC 气垫调整 AT %I11.0, 1 s
   "气垫快排" : Bool = PLC 气垫快排 AT %I14.2, 1 s
   "气垫向上" : Bool = PLC 气垫向上 AT %I14.4, 1 s
   "气垫向下" : Bool = PLC 气垫向下 AT %I14.5, 1 s
   "气垫向上(2)" : Bool = PLC "气垫向上(2)" AT %Q2.7, 1 s
   "气垫向下(2)" : Bool = PLC "气垫向下(2)" AT %Q3.0, 1 s
   "气垫快排阀" : Bool = PLC 气垫快排阀 AT %Q12.7, 1 s
   "滑块空开" : Bool = PLC 滑块空开 AT %I3.3, 1 s
   "滑块调整" : Bool = PLC 滑块调整 AT %I11.1, 1 s
   "滑块调整条件" : Bool = PLC 滑块调整条件 AT %M330.0, 1 s
   "滑块上限" : Bool = PLC 滑块上限 AT %I22.7, 1 s
   "滑块软限位上" : Bool = PLC 滑块软限位上 AT %M15.5, 1 s
   "滑块调整自动向上" : Bool = PLC 滑块调整自动向上 AT %M16.0, 1 s
   "滑块调整自动向下" : Bool = PLC 滑块调整自动向下 AT %M16.1, 1 s
   "滑块下限" : Bool = PLC 滑块下限 AT %I23.0, 1 s
   "滑块软限位下" : Bool = PLC 滑块软限位下 AT %M15.6, 1 s
   "模具更换" : Bool = PLC 模具更换 AT %I11.3, 1 s
   "急停故障" : Bool = PLC 急停故障 AT %M6.0, 1 s
   "液压保护气动泵阀" : Bool = PLC 液压保护气动泵阀 AT %Q12.6, 1 s
   "润滑检测2" : Bool = PLC 润滑检测2 AT %I20.1, 100 ms
   "计数清零" : Bool = PLC 计数清零 AT %M20.1, 1 s
   "计数开始" : Bool = PLC 计数开始 AT %M20.0, 1 s
   "断电保持数据_目标产量" : Int = PLC 断电保持数据.目标产量, 1 s
   "断电保持数据_当前产量" : Int = PLC 断电保持数据.当前产量, 1 s
   "产量完成" : Bool = PLC 产量完成 AT %M800.0, 1 s
   "润滑故障" : Bool = PLC 润滑故障 AT %M500.0, 1 s

screen "工作台操作" 800x477
   TextField "文本域_1" at 47,79 size 125x27; Text '工作台松开'
   TextField "文本域_2" at 53,142 size 125x27; Text '工作台夹紧'
   Circle "圆_5" at 541,81 size 27x27
      Appearance <- "工作台放松阀(1)"
   TextField "文本域_10" at 513,111 size 83x16; Text '工作台松开阀'
   Circle "圆_7" at 469,81 size 27x27
      Appearance <- "工作台松开"
   TextField "文本域_12" at 446,111 size 70x16; Text '工作台松开'
   Circle "圆_8" at 289,81 size 27x27
      Appearance <- "上死点指示"
   TextField "文本域_13" at 282,111 size 44x16; Text '上死点'
   Circle "圆_9" at 630,81 size 27x27
      Appearance <- "工作台放松压检"
   TextField "文本域_14" at 597,111 size 96x16; Text '工作台松开压力'
   Circle "圆_6" at 718,81 size 27x27
      Appearance <- "工作台放松OK"
   TextField "文本域_11" at 693,111 size 84x16; Text '工作台松开OK'
   TextField "文本域_19" at 447,171 size 70x16; Text '工作台夹紧'
   Circle "圆_15" at 290,141 size 27x27
      Appearance <- "工作台落到位前"
   TextField "文本域_20" at 260,171 size 96x16; Text '工作台前落到位'
   Circle "圆_16" at 536,141 size 27x27
      Appearance <- "工作台夹紧阀(1)"
   TextField "文本域_21" at 515,171 size 83x16; Text '工作台夹紧阀'
   Circle "圆_1" at 632,141 size 27x27
      Appearance <- "工作台夹紧压检"
   TextField "文本域_3" at 599,171 size 96x16; Text '工作台夹紧压力'
   Circle "圆_2" at 721,141 size 27x27
      Appearance <- "工作台-夹紧OK"
   TextField "文本域_4" at 696,171 size 84x16; Text '工作台夹紧OK'
   Circle "圆_3" at 391,82 size 27x27
      Appearance <- "气垫落到位"
   TextField "文本域_5" at 374,111 size 70x16; Text '气垫落到位'
   Circle "圆_4" at 392,140 size 27x27
      Appearance <- "工作台落到位后"
   TextField "文本域_6" at 355,171 size 96x16; Text '工作台后落到位'
   Button "按钮_1" at 26,411 size 67x56; TextOn '滑块角度'; TextOff '滑块角度'
      on Click: ActivateScreen("滑块角度", 0)
   Button "按钮_2" at 95,411 size 67x56; TextOn '设备状态'; TextOff '设备状态'
      on Click: ActivateScreen("设备状态", 0)
   Button "按钮_3" at 163,411 size 71x57; TextOn '工作台操作'; TextOff '工作台操作'
      on Click: ActivateScreen("工作台操作", 0)
   Button "按钮_4" at 235,411 size 69x57; TextOn '气垫操作'; TextOff '气垫操作'
      on Click: ActivateScreen("气垫操作", 0)
   Button "按钮_5" at 306,411 size 66x57; TextOn '故障显示'; TextOff '故障显示'
      on Click: ActivateScreen("故障显示", 0)
   Button "按钮_8" at 375,411 size 68x59; TextOn '滑块调整'; TextOff '滑块调整'
      on Click: ActivateScreen("滑块调整", 0)
   Circle "圆_10" at 468,140 size 27x27
      Appearance <- "工作台松开"
   Circle "圆_11" at 211,82 size 27x27
      Appearance <- "模具更换"
   TextField "文本域_7" at 204,112 size 57x16; Text '模具更换'
   Circle "圆_12" at 210,141 size 27x27
      Appearance <- "模具更换"
   TextField "文本域_8" at 203,171 size 57x16; Text '模具更换'

screen "故障显示" 800x477
   Button "按钮_1" at 26,411 size 67x56; TextOn '滑块角度'; TextOff '滑块角度'
      on Click: ActivateScreen("滑块角度", 0)
   Button "按钮_2" at 95,411 size 67x56; TextOn '设备状态'; TextOff '设备状态'
      on Click: ActivateScreen("设备状态", 0)
   Button "按钮_3" at 163,411 size 71x57; TextOn '工作台操作'; TextOff '工作台操作'
      on Click: ActivateScreen("工作台操作", 0)
   Button "按钮_4" at 235,411 size 69x57; TextOn '气垫操作'; TextOff '气垫操作'
      on Click: ActivateScreen("气垫操作", 0)
   Button "按钮_5" at 306,411 size 66x57; TextOn '故障显示'; TextOff '故障显示'
      on Click: ActivateScreen("故障显示", 0)
   Button "按钮_8" at 374,411 size 68x59; TextOn '滑块调整'; TextOff '滑块调整'
      on Click: ActivateScreen("滑块调整", 0)

screen "气垫操作" 800x477
   TextField "文本域_1" at 55,82 size 101x27; Text '气垫上调'
   TextField "文本域_2" at 58,142 size 101x27; Text '气垫下调'
   Circle "圆_8" at 222,81 size 27x27
      Appearance <- "上死点"
   TextField "文本域_13" at 215,111 size 44x16; Text '上死点'
   Circle "圆_3" at 289,82 size 27x27
      Appearance <- "气垫落到位"
   TextField "文本域_5" at 268,112 size 70x16; Text '气垫落到位'
   Circle "圆_1" at 223,146 size 27x27
      Appearance <- "上死点"
   TextField "文本域_3" at 216,176 size 44x16; Text '上死点'
   Circle "圆_2" at 290,147 size 27x27
      Appearance <- "气垫落到位"
   TextField "文本域_4" at 269,177 size 70x16; Text '气垫落到位'
   Circle "圆_4" at 356,81 size 27x27
      Appearance <- "气垫上限"
   TextField "文本域_6" at 335,112 size 57x16; Text '气垫上限'
   Circle "圆_5" at 357,146 size 27x27
      Appearance <- "气垫下限"
   TextField "文本域_7" at 336,177 size 57x16; Text '气垫下限'
   Circle "圆_6" at 416,81 size 27x27
      Appearance <- "气垫调整空开"
   TextField "文本域_8" at 400,112 size 57x16; Text '气垫空开'
   Circle "圆_7" at 417,146 size 27x27
      Appearance <- "气垫调整空开"
   TextField "文本域_9" at 401,177 size 57x16; Text '气垫空开'
   Circle "圆_9" at 476,81 size 27x27
      Appearance <- "气垫调整"
   TextField "文本域_10" at 460,112 size 57x16; Text '气垫调整'
   Circle "圆_10" at 477,146 size 27x27
      Appearance <- "气垫调整"
   TextField "文本域_11" at 460,177 size 57x16; Text '气垫调整'
   Circle "圆_11" at 536,81 size 27x27
      Appearance <- "气垫快排"
   TextField "文本域_12" at 520,112 size 57x16; Text '气垫快排'
   Circle "圆_12" at 537,146 size 27x27
      Appearance <- "气垫快排"
   TextField "文本域_14" at 522,177 size 57x16; Text '气垫快排'
   Circle "圆_13" at 599,81 size 27x27
      Appearance <- "气垫向上"
   TextField "文本域_15" at 586,112 size 57x16; Text '气垫上调'
   Circle "圆_14" at 599,146 size 27x27
      Appearance <- "气垫向下"
   TextField "文本域_16" at 587,177 size 57x16; Text '气垫下调'
   Circle "圆_15" at 662,81 size 27x27
      Appearance <- "气垫向上(2)"
   TextField "文本域_17" at 652,112 size 44x16; Text '气垫上'
   Circle "圆_16" at 663,146 size 27x27
      Appearance <- "气垫向下(2)"
   TextField "文本域_18" at 652,177 size 44x16; Text '气垫下'
   TextField "文本域_19" at 58,210 size 101x27; Text '气垫快排'
   Circle "圆_17" at 223,214 size 27x27
      Appearance <- "上死点"
   TextField "文本域_20" at 216,244 size 44x16; Text '上死点'
   Circle "圆_18" at 311,215 size 27x27
      Appearance <- "工作台落到位后"
   TextField "文本域_21" at 267,244 size 96x16; Text '工作台后落到位'
   Circle "圆_19" at 400,214 size 27x27
      Appearance <- "工作台落到位前"
   TextField "文本域_22" at 364,243 size 96x16; Text '工作台前落到位'
   Circle "圆_20" at 488,213 size 27x27
      Appearance <- "气垫调整"
   TextField "文本域_23" at 471,244 size 57x16; Text '气垫调整'
   Circle "圆_21" at 576,213 size 27x27
      Appearance <- "气垫快排"
   TextField "文本域_24" at 559,244 size 57x16; Text '气垫快排'
   Circle "圆_22" at 661,214 size 27x27
      Appearance <- "气垫快排阀"
   TextField "文本域_25" at 646,245 size 70x16; Text '气垫快排阀'
   Button "按钮_1" at 26,411 size 67x56; TextOn '滑块角度'; TextOff '滑块角度'
      on Click: ActivateScreen("滑块角度", 0)
   Button "按钮_2" at 95,411 size 67x56; TextOn '设备状态'; TextOff '设备状态'
      on Click: ActivateScreen("设备状态", 0)
   Button "按钮_3" at 163,411 size 71x57; TextOn '工作台操作'; TextOff '工作台操作'
      on Click: ActivateScreen("工作台操作", 0)
   Button "按钮_4" at 235,411 size 69x57; TextOn '气垫操作'; TextOff '气垫操作'
      on Click: ActivateScreen("气垫操作", 0)
   Button "按钮_5" at 306,411 size 66x57; TextOn '故障显示'; TextOff '故障显示'
      on Click: ActivateScreen("故障显示", 0)
   Button "按钮_8" at 373,411 size 68x59; TextOn '滑块调整'; TextOff '滑块调整'
      on Click: ActivateScreen("滑块调整", 0)

screen "滑块角度" 800x477
   Circle "圆_2" at 245,51 size 21x21
      Appearance <- "360"
   Circle "圆_3" at 274,56 size 21x21
      Appearance <- "10度"
   Circle "圆_4" at 303,66 size 21x21
      Appearance <- "20度"
   Circle "圆_5" at 326,79 size 21x21
      Appearance <- "30度"
   Circle "圆_6" at 346,95 size 21x21
      Appearance <- "40度"
   Circle "圆_7" at 364,115 size 21x21
      Appearance <- "50"
   Circle "圆_8" at 377,135 size 21x21
      Appearance <- "60"
   Circle "圆_9" at 385,157 size 21x21
      Appearance <- "70"
   Circle "圆_10" at 392,179 size 21x21
      Appearance <- "80"
   Circle "圆_11" at 394,202 size 21x21
      Appearance <- "90"
   Circle "圆_12" at 391,226 size 21x21
      Appearance <- "100"
   Circle "圆_13" at 386,249 size 21x21
      Appearance <- "110"
   Circle "圆_14" at 378,271 size 21x21
      Appearance <- "120"
   Circle "圆_15" at 365,292 size 21x21
      Appearance <- "130"
   Circle "圆_16" at 348,311 size 21x21
      Appearance <- "140"
   Circle "圆_17" at 328,328 size 21x21
      Appearance <- "150"
   Circle "圆_18" at 306,342 size 21x21
      Appearance <- "160"
   Circle "圆_19" at 276,353 size 21x21
      Appearance <- "170"
   Circle "圆_20" at 247,357 size 21x21
      Appearance <- "180"
   Circle "圆_22" at 219,352 size 21x21
      Appearance <- "190"
   Circle "圆_23" at 195,344 size 21x21
      Appearance <- "200"
   Circle "圆_24" at 172,333 size 21x21
      Appearance <- "210"
   Circle "圆_25" at 152,319 size 21x21
      Appearance <- "220"
   Circle "圆_26" at 133,302 size 21x21
      Appearance <- "230"
   Circle "圆_27" at 117,281 size 21x21
      Appearance <- "240"
   Circle "圆_28" at 104,258 size 21x21
      Appearance <- "250"
   Circle "圆_29" at 96,229 size 21x21
      Appearance <- "260"
   Circle "圆_30" at 93,201 size 21x21
      Appearance <- "270"
   Circle "圆_32" at 95,178 size 21x21
      Appearance <- "280"
   Circle "圆_33" at 100,155 size 21x21
      Appearance <- "290"
   Circle "圆_34" at 110,131 size 21x21
      Appearance <- "300"
   Circle "圆_35" at 126,111 size 21x21
      Appearance <- "310"
   Circle "圆_36" at 144,91 size 21x21
      Appearance <- "320"
   Circle "圆_37" at 167,74 size 21x21
      Appearance <- "330"
   Circle "圆_38" at 191,63 size 21x21
      Appearance <- "340"
   Circle "圆_39" at 218,54 size 21x21
      Appearance <- "350"
   TextField "文本域_2" at 422,193 size 43x40; Text '90'
   TextField "文本域_3" at 221,378 size 62x40; Text '180'
   TextField "文本域_5" at 196,118 size 117x31; Text '滑块位置'
   TextField "文本域_4" at 25,203 size 62x40; Text '270'
   TextField "文本域_1" at 241,12 size 24x40; Text '0'
   SymbolLibrary "符号库_1" at 544,25 size 109x71
   SymbolLibrary "符号库_2" at 680,47 size 86x40
   TextField "文本域_7" at 671,101 size 77x21; Text '滑块电机'
   TextField "文本域_6" at 562,103 size 59x21; Text '主电机'
   TextField "文本域_8" at 487,149 size 93x25; Text '目标产量'
   Circle "圆_1" at 582,59 size 22x22
      Appearance <- "主电机运行指示"
   TextField "文本域_11" at 506,333 size 93x25; Text '润滑检测'
   Circle "圆_21" at 687,27 size 14x14
      Appearance <- "滑块向上KM6"
   Circle "圆_31" at 729,27 size 14x14
      Appearance <- "滑块向下KM7"
   TextField "文本域_15" at 677,7 size 33x17; Text '向上'
   TextField "文本域_16" at 719,8 size 33x17; Text '向下'
   Button "按钮_1" at 28,417 size 67x56; TextOn '滑块角度'; TextOff '滑块角度'
      on Click: ActivateScreen("滑块角度", 0)
   Button "按钮_2" at 96,417 size 67x56; TextOn '设备状态'; TextOff '设备状态'
      on Click: ActivateScreen("设备状态", 0)
   Button "按钮_3" at 163,417 size 71x55; TextOn '工作台操作'; TextOff '工作台操作'
      on Click: ActivateScreen("工作台操作", 0)
   Button "按钮_4" at 235,417 size 69x56; TextOn '气垫操作'; TextOff '气垫操作'
      on Click: ActivateScreen("气垫操作", 0)
   Button "按钮_5" at 304,416 size 66x57; TextOn '故障显示'; TextOff '故障显示'
      on Click: ActivateScreen("故障显示", 0)
   IOField "I/O 域_1" at 228,153 size 56x32; FormatPattern 999
      ProcessValue <- "横梁编码器 _DB_0.11"
   Button "按钮_8" at 373,416 size 68x56; TextOn '滑块调整'; TextOff '滑块调整'
      on Click: ActivateScreen("滑块调整", 0)
   IOField "I/O 域_2" at 487,180 size 83x38; FormatPattern 9999
      ProcessValue <- "断电保持数据_目标产量"
   TextField "文本域_14" at 487,230 size 93x25; Text '当前产量'
   Button "按钮_11" at 726,149 size 65x68; TextOff '计数清零'
      Appearance <- "ECamdata _DB_D102"
      on Press: SetBit("计数清零")
      on Release: ResetBit("计数清零")
   Circle "圆_42" at 532,374 size 48x48
      Appearance <- "润滑检测2"
   Switch "开关_1" at 597,136 size 120x88; CaptionText '计数通断'; TextOff '计数断'; TextOn '计数通'
      on SwitchOn: SetBit("计数开始")
      on SwitchOff: ResetBit("计数开始")
      ProcessValue <- "计数开始"
   IOField "I/O 域_4" at 487,256 size 83x38; FormatPattern 9999
      ProcessValue <- "断电保持数据_当前产量"
   TextField "文本域_10" at 585,256 size 153x40; Text '产量完成'
      Appearance <- "产量完成"
   Circle "圆_43" at 674,374 size 48x48
      Appearance <- "润滑故障"
   TextField "文本域_9" at 650,333 size 93x25; Text '润滑故障'

screen "滑块调整" 800x477
   Button "按钮_1" at 26,411 size 67x56; TextOn '滑块角度'; TextOff '滑块角度'
      on Click: ActivateScreen("滑块角度", 0)
   Button "按钮_2" at 95,411 size 67x56; TextOn '设备状态'; TextOff '设备状态'
      on Click: ActivateScreen("设备状态", 0)
   Button "按钮_3" at 163,411 size 71x57; TextOn '工作台操作'; TextOff '工作台操作'
      on Click: ActivateScreen("工作台操作", 0)
   Button "按钮_4" at 235,411 size 69x57; TextOn '气垫操作'; TextOff '气垫操作'
      on Click: ActivateScreen("气垫操作", 0)
   Button "按钮_5" at 306,411 size 66x57; TextOn '故障显示'; TextOff '故障显示'
      on Click: ActivateScreen("故障显示", 0)
   Button "按钮_8" at 374,411 size 68x59; TextOn '滑块调整'; TextOff '滑块调整'
      on Click: ActivateScreen("滑块调整", 0)
   TextField "文本域_1" at 157,34 size 61x29; Text '1200'
   TextField "文本域_2" at 26,34 size 109x29; Text '滑块上限'
   TextField "文本域_3" at 158,114 size 47x29; Text '600'
   TextField "文本域_4" at 27,114 size 109x29; Text '滑块下限'
   TextField "文本域_6" at 236,33 size 135x29; Text '滑块当前值'
   TextField "文本域_8" at 240,108 size 135x29; Text '滑块设定值'
   Circle "圆_1" at 579,39 size 52x52
      Appearance <- "滑块调整手动/自动"
   Circle "圆_2" at 683,40 size 53x53
      Appearance <- "滑块调整手动/自动"
   TextField "文本域_16" at 583,117 size 41x21; Text '手动'
   TextField "文本域_19" at 689,116 size 41x21; Text '自动'
   IOField "I/O 域_1" at 382,97 size 136x47; FormatPattern 9999
      ProcessValue <- "横梁编码器 _DB_+0.8"
   IOField "I/O 域_2" at 377,33 size 140x47; FormatPattern 9999
      ProcessValue <- "ECamdata _DB_D107"
   TextField "文本域_7" at 0,0 size 125x30; Text '滑块调整手动/自动'
   TextField "文本域_5" at 0,0 size 125x30; Text '滑块调整手动/自动'
   TextField "文本域_10" at 0,0 size 125x30; Text '滑块调整手动/自动'
   TextField "文本域_9" at 44,162 size 149x27; Text '滑块调整条件'
   Circle "圆_8" at 222,161 size 27x27
      Appearance <- "上死点"
   TextField "文本域_13" at 215,191 size 44x16; Text '上死点'
   Circle "圆_3" at 289,162 size 27x27
      Appearance <- "平衡缸气压检测"
   TextField "文本域_11" at 268,192 size 70x16; Text '平衡缸压力'
   Circle "圆_4" at 347,161 size 27x27
      Appearance <- "滑块空开"
   TextField "文本域_14" at 338,192 size 57x16; Text '滑块空开'
   Circle "圆_9" at 414,161 size 27x27
      Appearance <- "液压保护压力检测"
   TextField "文本域_15" at 398,192 size 83x16; Text '液压保护压力'
   Circle "圆_13" at 497,161 size 27x27
      Appearance <- "滑块调整"
   TextField "文本域_18" at 484,192 size 57x16; Text '滑块调整'
   Circle "圆_15" at 565,161 size 27x27
      Appearance <- "滑块调整条件"
   TextField "文本域_20" at 546,192 size 83x16; Text '滑块调整条件'
   TextField "文本域_12" at 65,269 size 101x27; Text '滑块调整'
   Circle "圆_5" at 300,276 size 27x27
      Appearance <- "滑块向上"
   TextField "文本域_17" at 293,306 size 44x16; Text '滑块上'
   Circle "圆_6" at 348,248 size 27x27
      Appearance <- "滑块调整手动/自动"
   TextField "文本域_21" at 333,278 size 57x16; Text '滑块手动'
   Circle "圆_7" at 444,254 size 27x27
      Appearance <- "滑块上限"
   TextField "文本域_22" at 435,285 size 57x16; Text '滑块上限'
   Circle "圆_10" at 500,254 size 27x27
      Appearance <- "滑块软限位上"
   TextField "文本域_23" at 492,285 size 44x16; Text '上软限'
   Circle "圆_11" at 549,254 size 27x27
      Appearance <- "滑块向上KM6"
   TextField "文本域_24" at 536,285 size 57x16; Text '滑块向上'
   Circle "圆_12" at 245,307 size 27x27
      Appearance <- "滑块调整条件"
   TextField "文本域_25" at 217,338 size 83x16; Text '滑块调整条件'
   Circle "圆_16" at 349,307 size 27x27
      Appearance <- "滑块调整手动/自动"
   TextField "文本域_27" at 334,337 size 57x16; Text '滑块自动'
   Circle "圆_14" at 394,280 size 27x27
      Appearance <- "滑块调整自动向上"
   TextField "文本域_26" at 379,310 size 57x16; Text '自动向上'
   Circle "圆_17" at 397,327 size 27x27
      Appearance <- "滑块调整自动向下"
   TextField "文本域_28" at 382,357 size 57x16; Text '自动向下'
   Circle "圆_18" at 447,343 size 27x27
      Appearance <- "滑块下限"
   TextField "文本域_29" at 438,374 size 57x16; Text '滑块下限'
   Circle "圆_19" at 503,343 size 27x27
      Appearance <- "滑块软限位下"
   TextField "文本域_30" at 495,374 size 44x16; Text '下软限'
   Circle "圆_20" at 552,343 size 27x27
      Appearance <- "滑块向下KM7"
   TextField "文本域_31" at 539,374 size 57x16; Text '滑块向下'
   Circle "圆_21" at 351,361 size 27x27
      Appearance <- "滑块调整手动/自动"
   TextField "文本域_32" at 336,391 size 57x16; Text '滑块手动'
   Circle "圆_22" at 301,333 size 27x27
      Appearance <- "滑块向上"
   TextField "文本域_33" at 294,363 size 44x16; Text '滑块下'
   Button "按钮_6" at 82,249 size 192x32; TextOff '滑块调整'
      on Click: ActivateScreen("滑块调整", 0)

screen "设备状态" 800x477
   TextField "文本域_1" at 63,79 size 101x27; Text '润滑正常'
   TextField "文本域_2" at 64,142 size 101x27; Text '急停正常'
   TextField "文本域_3" at 50,205 size 125x27; Text '工作台夹紧'
   TextField "文本域_4" at 66,268 size 101x27; Text '气压正常'
   TextField "文本域_5" at 46,331 size 149x27; Text '液压保护正常'
   Circle "圆_1" at 325,208 size 27x27
      Appearance <- "工作台落到位前"
   TextField "文本域_6" at 293,237 size 96x16; Text '工作台前落到位'
   Circle "圆_2" at 427,207 size 27x27
      Appearance <- "工作台落到位后"
   TextField "文本域_7" at 395,237 size 96x16; Text '工作台后落到位'
   Circle "圆_3" at 527,207 size 27x27
      Appearance <- "工作台夹紧压检"
   TextField "文本域_8" at 495,237 size 96x16; Text '工作台夹紧压力'
   Circle "圆_4" at 223,207 size 27x27
      Appearance <- "工作台夹紧阀(1)"
   TextField "文本域_9" at 198,237 size 83x16; Text '工作台夹紧阀'
   Circle "圆_5" at 427,81 size 27x27
      Appearance <- "润滑油压正常"
   TextField "文本域_10" at 399,111 size 83x16; Text '润滑油压正常'
   Circle "圆_7" at 325,81 size 27x27
      Appearance <- "滤油器堵塞指示"
   TextField "文本域_12" at 295,111 size 96x16; Text '润滑过滤器正常'
   Circle "圆_8" at 222,81 size 27x27
      Appearance <- "工作台落到位后"
   TextField "文本域_13" at 196,111 size 83x16; Text '润滑油位正常'
   Circle "圆_9" at 527,81 size 27x27
      Appearance <- "工作台落到位后"
   TextField "文本域_14" at 502,111 size 83x16; Text '润滑频次正常'
   Circle "圆_10" at 325,270 size 27x27
      Appearance <- "工作台落到位前"
   TextField "文本域_15" at 306,299 size 70x16; Text '离合器压力'
   Circle "圆_11" at 427,269 size 27x27
      Appearance <- "工作台落到位后"
   Circle "圆_12" at 223,269 size 27x27
      Appearance <- "平衡缸气压检测"
   TextField "文本域_16" at 200,298 size 70x16; Text '平衡缸压力'
   TextField "文本域_17" at 407,300 size 70x16; Text '制动器压力'
   Circle "圆_6" at 615,81 size 27x27
      Appearance <- "润滑油泵启动OK"
   TextField "文本域_11" at 590,111 size 83x16; Text '润滑电机启动'
   Circle "圆_14" at 325,141 size 27x27
      Appearance <- "急停故障"
   TextField "文本域_19" at 312,171 size 57x16; Text '急停闭点'
   Circle "圆_15" at 222,141 size 27x27
      Appearance <- "急停开点左前"
   TextField "文本域_20" at 207,171 size 57x16; Text '急停开点'
   Circle "圆_16" at 428,141 size 27x27
      Appearance <- "爬梯开关"
   TextField "文本域_21" at 414,171 size 57x16; Text '梯子开关'
   Circle "圆_18" at 325,333 size 27x27
      Appearance <- "液压保护卸荷"
   TextField "文本域_23" at 306,362 size 70x16; Text '卸荷阀卸荷'
   Circle "圆_19" at 427,332 size 27x27
      Appearance <- "液压保护卸荷"
   Circle "圆_20" at 223,332 size 27x27
      Appearance <- "液压保护压力检测"
   TextField "文本域_24" at 200,361 size 83x16; Text '液压保护压力'
   TextField "文本域_25" at 415,364 size 44x16; Text '气源阀'
   Button "按钮_1" at 26,411 size 67x56; TextOn '滑块角度'; TextOff '滑块角度'
      on Click: ActivateScreen("滑块角度", 0)
   Button "按钮_2" at 95,411 size 67x56; TextOn '设备状态'; TextOff '设备状态'
      on Click: ActivateScreen("设备状态", 0)
   Button "按钮_3" at 163,411 size 71x57; TextOn '工作台操作'; TextOff '工作台操作'
      on Click: ActivateScreen("工作台操作", 0)
   Button "按钮_4" at 235,411 size 69x57; TextOn '气垫操作'; TextOff '气垫操作'
      on Click: ActivateScreen("气垫操作", 0)
   Button "按钮_5" at 306,411 size 66x57; TextOn '故障显示'; TextOff '故障显示'
      on Click: ActivateScreen("故障显示", 0)
   Button "按钮_8" at 374,411 size 68x59; TextOn '滑块调整'; TextOff '滑块调整'
      on Click: ActivateScreen("滑块调整", 0)
   Circle "圆_13" at 493,332 size 27x27
      Appearance <- "液压保护气动泵阀"
   TextField "文本域_18" at 481,363 size 57x16; Text '气动泵阀'
*)